LIN {X 0,Y 573.521,Z 573.892,A -85,B 0,C 180,E1 -2263.87,E2 -2263.87} C_VEL
LIN {X 0,Y 573.779,Z 548.951,A -85,B 0,C 180,E1 -2266.545,E2 -2266.545} C_VEL
LIN {X 0,Y 574.092,Z 520.138,A -85,B 0,C 180,E1 -2269.699,E2 -2269.699} C_VEL
LIN {X 0,Y 574.414,Z 495.16,A -85,B 0,C 180,E1 -2272.479,E2 -2272.479} C_VEL
LIN {X 0,Y 574.81,Z 471.063,A -85,B 0,C 180,E1 -2275.207,E2 -2275.207} C_VEL
LIN {X 0,Y 574.89,Z 460.282,A -85,B 0,C 180,E1 -2276.409,E2 -2276.409} C_VEL
LIN {X 0,Y 573.276,Z 453.235,A -85,B 0,C 180,E1 -2277.27,E2 -2277.27} C_VEL
LIN {X 0,Y 573.249,Z 453.075,A -85,B 0,C 180,E1 -2280.175,E2 -2280.175} C_VEL
LIN {X 0,Y 573.254,Z 453.074,A -85,B 0,C 180,E1 -2282.644,E2 -2282.644} C_VEL
LIN {X 0,Y 573.205,Z 453.079,A -85,B 0,C 180,E1 -2285.187,E2 -2285.187} C_VEL
LIN {X 0,Y 573.234,Z 453.078,A -85,B 0,C 180,E1 -2287.807,E2 -2287.807} C_VEL
LIN {X 0,Y 573.266,Z 453.074,A -85,B 0,C 180,E1 -2290.527,E2 -2290.527} C_VEL
LIN {X 0,Y 573.249,Z 453.075,A -85,B 0,C 180,E1 -2293.669,E2 -2293.669} C_VEL
LIN {X 0,Y 573.234,Z 453.076,A -85,B 0,C 180,E1 -2296.64,E2 -2296.64} C_VEL
LIN {X 0,Y 573.268,Z 453.071,A -85,B 0,C 180,E1 -2299.477,E2 -2299.477} C_VEL
LIN {X 0,Y 573.23,Z 453.083,A -85,B 0,C 180,E1 -2302.192,E2 -2302.192} C_VEL
LIN {X 0,Y 573.263,Z 453.073,A -85,B 0,C 180,E1 -2304.816,E2 -2304.816} C_VEL
LIN {X 0,Y 573.249,Z 453.071,A -85,B 0,C 180,E1 -2307.355,E2 -2307.355} C_VEL
LIN {X 0,Y 573.249,Z 453.075,A -85,B 0,C 180,E1 -2309.824,E2 -2309.824} C_VEL
LIN {X 0,Y 573.281,Z 453.076,A -85,B 0,C 180,E1 -2312.235,E2 -2312.235} C_VEL
LIN {X 0,Y 573.261,Z 453.071,A -85,B 0,C 180,E1 -2315.12,E2 -2315.12} C_VEL
LIN {X 0,Y 573.23,Z 453.076,A -85,B 0,C 180,E1 -2317.662,E2 -2317.662} C_VEL
LIN {X 0,Y 573.248,Z 453.073,A -85,B 0,C 180,E1 -2319.923,E2 -2319.923} C_VEL
LIN {X 0,Y 573.253,Z 453.073,A -85,B 0,C 180,E1 -2322.988,E2 -2322.988} C_VEL
LIN {X 0,Y 573.263,Z 453.072,A -85,B 0,C 180,E1 -2325.807,E2 -2325.807} C_VEL
LIN {X 0,Y 573.273,Z 453.074,A -85,B 0,C 180,E1 -2328.734,E2 -2328.734} C_VEL
LIN {X 0,Y 573.298,Z 453.066,A -85,B 0,C 180,E1 -2331.541,E2 -2331.541} C_VEL
LIN {X 0,Y 573.285,Z 453.075,A -85,B 0,C 180,E1 -2334.372,E2 -2334.372} C_VEL
LIN {X 0,Y 573.3,Z 453.067,A -85,B 0,C 180,E1 -2337.892,E2 -2337.892} C_VEL
LIN {X 0,Y 573.33,Z 453.07,A -85,B 0,C 180,E1 -2340.702,E2 -2340.702} C_VEL
LIN {X 0,Y 573.233,Z 453.073,A -85,B 0,C 180,E1 -2343.515,E2 -2343.515} C_VEL
LIN {X 0,Y 573.29,Z 453.067,A -85,B 0,C 180,E1 -2345.628,E2 -2345.628} C_VEL
LIN {X 0,Y 573.299,Z 453.073,A -85,B 0,C 180,E1 -2348.459,E2 -2348.459} C_VEL
LIN {X 0,Y 573.289,Z 453.069,A -85,B 0,C 180,E1 -2351.312,E2 -2351.312} C_VEL
LIN {X 0,Y 573.271,Z 453.075,A -85,B 0,C 180,E1 -2354.425,E2 -2354.425} C_VEL
LIN {X 0,Y 573.251,Z 453.076,A -85,B 0,C 180,E1 -2357.112,E2 -2357.112} C_VEL
LIN {X 0,Y 573.249,Z 453.074,A -85,B 0,C 180,E1 -2360.077,E2 -2360.077} C_VEL
LIN {X 0,Y 573.231,Z 453.077,A -85,B 0,C 180,E1 -2362.338,E2 -2362.338} C_VEL
LIN {X 0,Y 573.244,Z 453.077,A -85,B 0,C 180,E1 -2364.403,E2 -2364.403} C_VEL
LIN {X 0,Y 572.618,Z 453.162,A -85,B 0,C 180,E1 -2364.99,E2 -2364.99} C_VEL
LIN {X 0,Y 569.779,Z 453.515,A -85,B 0,C 180,E1 -2365.942,E2 -2365.942} C_VEL
LIN {X 0,Y 567.35,Z 453.816,A -85,B 0,C 180,E1 -2366.708,E2 -2366.708} C_VEL
LIN {X 0,Y 566.298,Z 453.94,A -85,B 0,C 180,E1 -2367.299,E2 -2367.299} C_VEL
LIN {X 0,Y 566.209,Z 453.949,A -85,B 0,C 180,E1 -2367.499,E2 -2367.499} C_VEL
LIN {X 0,Y 566.187,Z 453.953,A -85,B 0,C 180,E1 -2370.593,E2 -2370.593} C_VEL
LIN {X 0,Y 566.222,Z 453.953,A -85,B 0,C 180,E1 -2373.102,E2 -2373.102} C_VEL
LIN {X 0,Y 566.208,Z 453.95,A -85,B 0,C 180,E1 -2375.689,E2 -2375.689} C_VEL
LIN {X 0,Y 566.212,Z 453.952,A -85,B 0,C 180,E1 -2378.56,E2 -2378.56} C_VEL
LIN {X 0,Y 566.207,Z 453.955,A -85,B 0,C 180,E1 -2381.137,E2 -2381.137} C_VEL
LIN {X 0,Y 566.196,Z 453.951,A -85,B 0,C 180,E1 -2384.036,E2 -2384.036} C_VEL
LIN {X 0,Y 566.207,Z 453.955,A -85,B 0,C 180,E1 -2387.083,E2 -2387.083} C_VEL
LIN {X 0,Y 566.225,Z 453.948,A -85,B 0,C 180,E1 -2389.804,E2 -2389.804} C_VEL
LIN {X 0,Y 566.198,Z 453.954,A -85,B 0,C 180,E1 -2392.6,E2 -2392.6} C_VEL
LIN {X 0,Y 566.212,Z 453.947,A -85,B 0,C 180,E1 -2395.183,E2 -2395.183} C_VEL
LIN {X 0,Y 566.234,Z 453.947,A -85,B 0,C 180,E1 -2397.745,E2 -2397.745} C_VEL
LIN {X 0,Y 566.204,Z 453.952,A -85,B 0,C 180,E1 -2400.329,E2 -2400.329} C_VEL
LIN {X 0,Y 566.212,Z 453.949,A -85,B 0,C 180,E1 -2402.662,E2 -2402.662} C_VEL
LIN {X 0,Y 566.238,Z 453.954,A -85,B 0,C 180,E1 -2405.04,E2 -2405.04} C_VEL
LIN {X 0,Y 566.196,Z 453.949,A -85,B 0,C 180,E1 -2408.138,E2 -2408.138} C_VEL
LIN {X 0,Y 566.239,Z 453.949,A -85,B 0,C 180,E1 -2410.612,E2 -2410.612} C_VEL
LIN {X 0,Y 566.218,Z 453.944,A -85,B 0,C 180,E1 -2413.413,E2 -2413.413} C_VEL
LIN {X 0,Y 566.282,Z 454.118,A -85,B 0,C 180,E1 -2416.293,E2 -2416.293} C_VEL
LIN {X 0,Y 566.5,Z 455.143,A -85,B 0,C 180,E1 -2416.407,E2 -2416.407} C_VEL
LIN {X 0,Y 567.065,Z 456.976,A -85,B 0,C 180,E1 -2416.453,E2 -2416.453} C_VEL
LIN {X 0,Y 566.992,Z 533.99,A -85,B 0,C 180,E1 -2417.45,E2 -2417.45} C_VEL
LIN {X 0,Y 566.878,Z 547.245,A -85,B 0,C 180,E1 -2417.765,E2 -2417.765} C_VEL
LIN {X 0,Y 566.749,Z 559.399,A -85,B 0,C 180,E1 -2418.194,E2 -2418.194} C_VEL
LIN {X 0,Y 566.633,Z 571.542,A -85,B 0,C 180,E1 -2418.776,E2 -2418.776} C_VEL
LIN {X 0,Y 566.459,Z 582.558,A -85,B 0,C 180,E1 -2419.456,E2 -2419.456} C_VEL
LIN {X 0,Y 566.323,Z 593.075,A -85,B 0,C 180,E1 -2420.266,E2 -2420.266} C_VEL
LIN {X 0,Y 566.221,Z 601.673,A -85,B 0,C 180,E1 -2421.075,E2 -2421.075} C_VEL
LIN {X 0,Y 566.113,Z 609.593,A -85,B 0,C 180,E1 -2421.972,E2 -2421.972} C_VEL
LIN {X 0,Y 566.05,Z 616.16,A -85,B 0,C 180,E1 -2422.868,E2 -2422.868} C_VEL
LIN {X 0,Y 566.003,Z 622.629,A -85,B 0,C 180,E1 -2423.942,E2 -2423.942} C_VEL
LIN {X 0,Y 565.878,Z 627.766,A -85,B 0,C 180,E1 -2425.013,E2 -2425.013} C_VEL
LIN {X 0,Y 565.926,Z 631.754,A -85,B 0,C 180,E1 -2426.084,E2 -2426.084} C_VEL
LIN {X 0,Y 565.877,Z 634.704,A -85,B 0,C 180,E1 -2427.153,E2 -2427.153} C_VEL
LIN {X 0,Y 565.84,Z 636.128,A -85,B 0,C 180,E1 -2427.865,E2 -2427.865} C_VEL
LIN {X 0,Y 565.841,Z 637.756,A -85,B 0,C 180,E1 -2429.288,E2 -2429.288} C_VEL
LIN {X 0,Y 565.839,Z 637.996,A -85,B 0,C 180,E1 -2430,E2 -2430} C_VEL
LIN {X 0,Y 565.841,Z 637.815,A -85,B 0,C 180,E1 -2430.712,E2 -2430.712} C_VEL
LIN {X 0,Y 565.84,Z 636.269,A -85,B 0,C 180,E1 -2432.135,E2 -2432.135} C_VEL
LIN {X 0,Y 565.878,Z 634.909,A -85,B 0,C 180,E1 -2432.847,E2 -2432.847} C_VEL
LIN {X 0,Y 565.927,Z 632.029,A -85,B 0,C 180,E1 -2433.916,E2 -2433.916} C_VEL
LIN {X 0,Y 565.878,Z 628.129,A -85,B 0,C 180,E1 -2434.987,E2 -2434.987} C_VEL
LIN {X 0,Y 565.99,Z 623.098,A -85,B 0,C 180,E1 -2436.058,E2 -2436.058} C_VEL
LIN {X 0,Y 566.031,Z 616.774,A -85,B 0,C 180,E1 -2437.132,E2 -2437.132} C_VEL
LIN {X 0,Y 566.133,Z 608.85,A -85,B 0,C 180,E1 -2438.207,E2 -2438.207} C_VEL
LIN {X 0,Y 566.249,Z 598.998,A -85,B 0,C 180,E1 -2439.285,E2 -2439.285} C_VEL
LIN {X 0,Y 566.423,Z 588.683,A -85,B 0,C 180,E1 -2440.184,E2 -2440.184} C_VEL
LIN {X 0,Y 566.581,Z 577.399,A -85,B 0,C 180,E1 -2440.971,E2 -2440.971} C_VEL
LIN {X 0,Y 566.679,Z 565.488,A -85,B 0,C 180,E1 -2441.626,E2 -2441.626} C_VEL
LIN {X 0,Y 566.819,Z 553.476,A -85,B 0,C 180,E1 -2442.122,E2 -2442.122} C_VEL
LIN {X 0,Y 566.936,Z 540.434,A -85,B 0,C 180,E1 -2442.506,E2 -2442.506} C_VEL
LIN {X 0,Y 567.025,Z 528.072,A -85,B 0,C 180,E1 -2442.732,E2 -2442.732} C_VEL
LIN {X 0,Y 566.994,Z 456.838,A -85,B 0,C 180,E1 -2443.64,E2 -2443.64} C_VEL
LIN {X 0,Y 566.421,Z 454.812,A -85,B 0,C 180,E1 -2443.704,E2 -2443.704} C_VEL
LIN {X 0,Y 566.255,Z 453.999,A -85,B 0,C 180,E1 -2443.845,E2 -2443.845} C_VEL
LIN {X 0,Y 566.227,Z 453.941,A -85,B 0,C 180,E1 -2447.113,E2 -2447.113} C_VEL
LIN {X 0,Y 566.214,Z 453.951,A -85,B 0,C 180,E1 -2449.58,E2 -2449.58} C_VEL
LIN {X 0,Y 566.195,Z 453.949,A -85,B 0,C 180,E1 -2451.862,E2 -2451.862} C_VEL
LIN {X 0,Y 566.219,Z 453.956,A -85,B 0,C 180,E1 -2455.029,E2 -2455.029} C_VEL
LIN {X 0,Y 566.212,Z 453.95,A -85,B 0,C 180,E1 -2457.338,E2 -2457.338} C_VEL
LIN {X 0,Y 566.202,Z 453.951,A -85,B 0,C 180,E1 -2459.768,E2 -2459.768} C_VEL
LIN {X 0,Y 566.206,Z 453.951,A -85,B 0,C 180,E1 -2462.43,E2 -2462.43} C_VEL
LIN {X 0,Y 566.199,Z 453.961,A -85,B 0,C 180,E1 -2464.992,E2 -2464.992} C_VEL
LIN {X 0,Y 566.195,Z 453.954,A -85,B 0,C 180,E1 -2467.46,E2 -2467.46} C_VEL
LIN {X 0,Y 566.225,Z 453.948,A -85,B 0,C 180,E1 -2470.196,E2 -2470.196} C_VEL
LIN {X 0,Y 566.202,Z 453.956,A -85,B 0,C 180,E1 -2473.053,E2 -2473.053} C_VEL
LIN {X 0,Y 566.194,Z 453.952,A -85,B 0,C 180,E1 -2476.048,E2 -2476.048} C_VEL
LIN {X 0,Y 566.207,Z 453.954,A -85,B 0,C 180,E1 -2478.863,E2 -2478.863} C_VEL
LIN {X 0,Y 566.185,Z 453.954,A -85,B 0,C 180,E1 -2481.637,E2 -2481.637} C_VEL
LIN {X 0,Y 566.208,Z 453.95,A -85,B 0,C 180,E1 -2484.311,E2 -2484.311} C_VEL
LIN {X 0,Y 566.222,Z 453.952,A -85,B 0,C 180,E1 -2486.898,E2 -2486.898} C_VEL
LIN {X 0,Y 566.187,Z 453.954,A -85,B 0,C 180,E1 -2489.407,E2 -2489.407} C_VEL
LIN {X 0,Y 566.22,Z 453.948,A -85,B 0,C 180,E1 -2491.858,E2 -2491.858} C_VEL
LIN {X 0,Y 566.219,Z 453.948,A -85,B 0,C 180,E1 -2494.251,E2 -2494.251} C_VEL
LIN {X 0,Y 566.184,Z 453.954,A -85,B 0,C 180,E1 -2496.713,E2 -2496.713} C_VEL
LIN {X 0,Y 566.212,Z 453.954,A -85,B 0,C 180,E1 -2499.663,E2 -2499.663} C_VEL
LIN {X 0,Y 566.195,Z 453.952,A -85,B 0,C 180,E1 -2502.668,E2 -2502.668} C_VEL
LIN {X 0,Y 566.223,Z 453.953,A -85,B 0,C 180,E1 -2505.626,E2 -2505.626} C_VEL
LIN {X 0,Y 566.265,Z 453.943,A -85,B 0,C 180,E1 -2508.654,E2 -2508.654} C_VEL
LIN {X 0,Y 566.241,Z 453.954,A -85,B 0,C 180,E1 -2511.434,E2 -2511.434} C_VEL
LIN {X 0,Y 566.252,Z 453.944,A -85,B 0,C 180,E1 -2514.302,E2 -2514.302} C_VEL
LIN {X 0,Y 566.271,Z 453.943,A -85,B 0,C 180,E1 -2517.866,E2 -2517.866} C_VEL
LIN {X 0,Y 566.298,Z 453.939,A -85,B 0,C 180,E1 -2520.711,E2 -2520.711} C_VEL
LIN {X 0,Y 566.271,Z 453.942,A -85,B 0,C 180,E1 -2522.846,E2 -2522.846} C_VEL
LIN {X 0,Y 566.252,Z 453.95,A -85,B 0,C 180,E1 -2525.698,E2 -2525.698} C_VEL
LIN {X 0,Y 566.239,Z 453.945,A -85,B 0,C 180,E1 -2528.566,E2 -2528.566} C_VEL
LIN {X 0,Y 566.241,Z 453.952,A -85,B 0,C 180,E1 -2531.454,E2 -2531.454} C_VEL
LIN {X 0,Y 566.223,Z 453.948,A -85,B 0,C 180,E1 -2534.507,E2 -2534.507} C_VEL
LIN {X 0,Y 566.195,Z 453.956,A -85,B 0,C 180,E1 -2537.332,E2 -2537.332} C_VEL
LIN {X 0,Y 566.211,Z 453.948,A -85,B 0,C 180,E1 -2540.337,E2 -2540.337} C_VEL
LIN {X 0,Y 566.181,Z 453.96,A -85,B 0,C 180,E1 -2543.404,E2 -2543.404} C_VEL
LIN {X 0,Y 566.218,Z 453.953,A -85,B 0,C 180,E1 -2545.749,E2 -2545.749} C_VEL
LIN {X 0,Y 566.199,Z 453.952,A -85,B 0,C 180,E1 -2548.204,E2 -2548.204} C_VEL
LIN {X 0,Y 566.186,Z 453.953,A -85,B 0,C 180,E1 -2550.593,E2 -2550.593} C_VEL
LIN {X 0,Y 566.222,Z 453.948,A -85,B 0,C 180,E1 -2553.102,E2 -2553.102} C_VEL
LIN {X 0,Y 566.207,Z 453.96,A -85,B 0,C 180,E1 -2555.689,E2 -2555.689} C_VEL
LIN {X 0,Y 566.21,Z 453.949,A -85,B 0,C 180,E1 -2558.56,E2 -2558.56} C_VEL
LIN {X 0,Y 566.206,Z 453.952,A -85,B 0,C 180,E1 -2561.137,E2 -2561.137} C_VEL
LIN {X 0,Y 566.192,Z 453.955,A -85,B 0,C 180,E1 -2564.036,E2 -2564.036} C_VEL
LIN {X 0,Y 566.201,Z 453.952,A -85,B 0,C 180,E1 -2567.083,E2 -2567.083} C_VEL
LIN {X 0,Y 566.224,Z 453.954,A -85,B 0,C 180,E1 -2569.804,E2 -2569.804} C_VEL
LIN {X 0,Y 566.197,Z 453.951,A -85,B 0,C 180,E1 -2572.6,E2 -2572.6} C_VEL
LIN {X 0,Y 566.205,Z 453.952,A -85,B 0,C 180,E1 -2575.183,E2 -2575.183} C_VEL
LIN {X 0,Y 566.233,Z 453.955,A -85,B 0,C 180,E1 -2577.744,E2 -2577.744} C_VEL
LIN {X 0,Y 566.203,Z 453.95,A -85,B 0,C 180,E1 -2580.329,E2 -2580.329} C_VEL
LIN {X 0,Y 566.238,Z 454.137,A -85,B 0,C 180,E1 -2582.563,E2 -2582.563} C_VEL
LIN {X 0,Y 568.003,Z 462.182,A -85,B 0,C 180,E1 -2583.55,E2 -2583.55} C_VEL
LIN {X 0,Y 567.78,Z 486.01,A -85,B 0,C 180,E1 -2586.194,E2 -2586.194} C_VEL
LIN {X 0,Y 567.361,Z 510.289,A -85,B 0,C 180,E1 -2588.948,E2 -2588.948} C_VEL
LIN {X 0,Y 566.973,Z 537.184,A -85,B 0,C 180,E1 -2591.948,E2 -2591.948} C_VEL
LIN {X 0,Y 566.679,Z 562.399,A -85,B 0,C 180,E1 -2594.72,E2 -2594.72} C_VEL
LIN {X 0,Y 566.56,Z 573.901,A -85,B 0,C 180,E1 -2595.956,E2 -2595.956} C_VEL
LIN {X 0,Y 567.212,Z 579.746,A -85,B 0,C 180,E1 -2596.064,E2 -2596.064} C_VEL
LIN {X 0,Y 566.975,Z 683.962,A -85,B 0,C 180,E1 -2597.404,E2 -2597.404} C_VEL
LIN {X 0,Y 566.891,Z 696.467,A -85,B 0,C 180,E1 -2597.697,E2 -2597.697} C_VEL
LIN {X 0,Y 566.745,Z 708.925,A -85,B 0,C 180,E1 -2598.13,E2 -2598.13} C_VEL
LIN {X 0,Y 566.627,Z 721.167,A -85,B 0,C 180,E1 -2598.709,E2 -2598.709} C_VEL
LIN {X 0,Y 566.459,Z 733.205,A -85,B 0,C 180,E1 -2599.456,E2 -2599.456} C_VEL
LIN {X 0,Y 566.319,Z 743.604,A -85,B 0,C 180,E1 -2600.266,E2 -2600.266} C_VEL
LIN {X 0,Y 566.207,Z 752.115,A -85,B 0,C 180,E1 -2601.074,E2 -2601.074} C_VEL
LIN {X 0,Y 566.112,Z 759.962,A -85,B 0,C 180,E1 -2601.972,E2 -2601.972} C_VEL
LIN {X 0,Y 566.003,Z 767.623,A -85,B 0,C 180,E1 -2603.047,E2 -2603.047} C_VEL
LIN {X 0,Y 566.004,Z 774.681,A -85,B 0,C 180,E1 -2604.299,E2 -2604.299} C_VEL
LIN {X 0,Y 565.933,Z 779.372,A -85,B 0,C 180,E1 -2605.37,E2 -2605.37} C_VEL
LIN {X 0,Y 565.927,Z 782.958,A -85,B 0,C 180,E1 -2606.44,E2 -2606.44} C_VEL
LIN {X 0,Y 565.878,Z 784.808,A -85,B 0,C 180,E1 -2607.153,E2 -2607.153} C_VEL
LIN {X 0,Y 565.846,Z 787.186,A -85,B 0,C 180,E1 -2608.577,E2 -2608.577} C_VEL
LIN {X 0,Y 565.839,Z 788,A -85,B 0,C 180,E1 -2610,E2 -2610} C_VEL
LIN {X 0,Y 565.846,Z 787.186,A -85,B 0,C 180,E1 -2611.423,E2 -2611.423} C_VEL
LIN {X 0,Y 565.878,Z 784.81,A -85,B 0,C 180,E1 -2612.847,E2 -2612.847} C_VEL
LIN {X 0,Y 565.926,Z 781.896,A -85,B 0,C 180,E1 -2613.916,E2 -2613.916} C_VEL
LIN {X 0,Y 565.878,Z 777.949,A -85,B 0,C 180,E1 -2614.987,E2 -2614.987} C_VEL
LIN {X 0,Y 566.002,Z 772.867,A -85,B 0,C 180,E1 -2616.058,E2 -2616.058} C_VEL
LIN {X 0,Y 566.04,Z 766.47,A -85,B 0,C 180,E1 -2617.132,E2 -2617.132} C_VEL
LIN {X 0,Y 566.133,Z 758.48,A -85,B 0,C 180,E1 -2618.207,E2 -2618.207} C_VEL
LIN {X 0,Y 566.228,Z 750.338,A -85,B 0,C 180,E1 -2619.105,E2 -2619.105} C_VEL
LIN {X 0,Y 566.339,Z 740.404,A -85,B 0,C 180,E1 -2620.005,E2 -2620.005} C_VEL
LIN {X 0,Y 566.526,Z 729.287,A -85,B 0,C 180,E1 -2620.807,E2 -2620.807} C_VEL
LIN {X 0,Y 566.66,Z 718.182,A -85,B 0,C 180,E1 -2621.445,E2 -2621.445} C_VEL
LIN {X 0,Y 566.743,Z 705.991,A -85,B 0,C 180,E1 -2621.988,E2 -2621.988} C_VEL
LIN {X 0,Y 566.903,Z 693.188,A -85,B 0,C 180,E1 -2622.393,E2 -2622.393} C_VEL
LIN {X 0,Y 566.991,Z 679.622,A -85,B 0,C 180,E1 -2622.664,E2 -2622.664} C_VEL
LIN {X 0,Y 567.072,Z 577.956,A -85,B 0,C 180,E1 -2623.962,E2 -2623.962} C_VEL
LIN {X 0,Y 566.566,Z 573.899,A -85,B 0,C 180,E1 -2624.043,E2 -2624.043} C_VEL
LIN {X 0,Y 566.841,Z 547.449,A -85,B 0,C 180,E1 -2626.919,E2 -2626.919} C_VEL
LIN {X 0,Y 567.214,Z 520.711,A -85,B 0,C 180,E1 -2629.883,E2 -2629.883} C_VEL
LIN {X 0,Y 567.67,Z 493.479,A -85,B 0,C 180,E1 -2632.953,E2 -2632.953} C_VEL
LIN {X 0,Y 567.919,Z 474.04,A -85,B 0,C 180,E1 -2635.135,E2 -2635.135} C_VEL
LIN {X 0,Y 567.848,Z 461.024,A -85,B 0,C 180,E1 -2636.584,E2 -2636.584} C_VEL
LIN {X 0,Y 566.228,Z 454.041,A -85,B 0,C 180,E1 -2637.463,E2 -2637.463} C_VEL
LIN {X 0,Y 566.187,Z 453.955,A -85,B 0,C 180,E1 -2640.592,E2 -2640.592} C_VEL
LIN {X 0,Y 566.219,Z 453.948,A -85,B 0,C 180,E1 -2643.101,E2 -2643.101} C_VEL
LIN {X 0,Y 566.16,Z 453.96,A -85,B 0,C 180,E1 -2645.691,E2 -2645.691} C_VEL
LIN {X 0,Y 566.214,Z 453.953,A -85,B 0,C 180,E1 -2648.558,E2 -2648.558} C_VEL
LIN {X 0,Y 566.208,Z 453.948,A -85,B 0,C 180,E1 -2651.135,E2 -2651.135} C_VEL
LIN {X 0,Y 566.196,Z 453.959,A -85,B 0,C 180,E1 -2654.035,E2 -2654.035} C_VEL
LIN {X 0,Y 566.196,Z 453.949,A -85,B 0,C 180,E1 -2657.082,E2 -2657.082} C_VEL
LIN {X 0,Y 566.221,Z 453.951,A -85,B 0,C 180,E1 -2659.802,E2 -2659.802} C_VEL
LIN {X 0,Y 566.192,Z 453.957,A -85,B 0,C 180,E1 -2662.598,E2 -2662.598} C_VEL
LIN {X 0,Y 566.215,Z 453.948,A -85,B 0,C 180,E1 -2665.182,E2 -2665.182} C_VEL
LIN {X 0,Y 566.228,Z 453.947,A -85,B 0,C 180,E1 -2667.743,E2 -2667.743} C_VEL
LIN {X 0,Y 566.221,Z 453.958,A -85,B 0,C 180,E1 -2670.323,E2 -2670.323} C_VEL
LIN {X 0,Y 566.226,Z 453.944,A -85,B 0,C 180,E1 -2673.334,E2 -2673.334} C_VEL
LIN {X 0,Y 566.19,Z 453.953,A -85,B 0,C 180,E1 -2675.819,E2 -2675.819} C_VEL
LIN {X 0,Y 566.208,Z 453.951,A -85,B 0,C 180,E1 -2678.902,E2 -2678.902} C_VEL
LIN {X 0,Y 566.204,Z 453.946,A -85,B 0,C 180,E1 -2681.172,E2 -2681.172} C_VEL
LIN {X 0,Y 566.212,Z 453.948,A -85,B 0,C 180,E1 -2683.412,E2 -2683.412} C_VEL
LIN {X 0,Y 566.191,Z 453.96,A -85,B 0,C 180,E1 -2686.359,E2 -2686.359} C_VEL
LIN {X 0,Y 566.265,Z 453.949,A -85,B 0,C 180,E1 -2688.654,E2 -2688.654} C_VEL
LIN {X 0,Y 566.239,Z 453.946,A -85,B 0,C 180,E1 -2691.434,E2 -2691.434} C_VEL
LIN {X 0,Y 566.253,Z 453.95,A -85,B 0,C 180,E1 -2694.302,E2 -2694.302} C_VEL
LIN {X 0,Y 566.272,Z 453.942,A -85,B 0,C 180,E1 -2697.866,E2 -2697.866} C_VEL
LIN {X 0,Y 566.3,Z 453.945,A -85,B 0,C 180,E1 -2700.711,E2 -2700.711} C_VEL
LIN {X 0,Y 566.272,Z 453.947,A -85,B 0,C 180,E1 -2702.846,E2 -2702.846} C_VEL
LIN {X 0,Y 566.258,Z 453.943,A -85,B 0,C 180,E1 -2705.698,E2 -2705.698} C_VEL
LIN {X 0,Y 566.24,Z 453.954,A -85,B 0,C 180,E1 -2708.566,E2 -2708.566} C_VEL
LIN {X 0,Y 566.241,Z 453.946,A -85,B 0,C 180,E1 -2711.454,E2 -2711.454} C_VEL
LIN {X 0,Y 566.224,Z 453.954,A -85,B 0,C 180,E1 -2714.507,E2 -2714.507} C_VEL
LIN {X 0,Y 566.195,Z 453.952,A -85,B 0,C 180,E1 -2717.332,E2 -2717.332} C_VEL
LIN {X 0,Y 566.212,Z 453.953,A -85,B 0,C 180,E1 -2720.337,E2 -2720.337} C_VEL
LIN {X 0,Y 566.182,Z 453.954,A -85,B 0,C 180,E1 -2723.404,E2 -2723.404} C_VEL
LIN {X 0,Y 566.219,Z 453.948,A -85,B 0,C 180,E1 -2725.749,E2 -2725.749} C_VEL
LIN {X 0,Y 566.209,Z 453.949,A -85,B 0,C 180,E1 -2727.499,E2 -2727.499} C_VEL
LIN {X 0,Y 565.531,Z 454.034,A -85,B 0,C 180,E1 -2728.093,E2 -2728.093} C_VEL
LIN {X 0,Y 562.667,Z 454.391,A -85,B 0,C 180,E1 -2729.057,E2 -2729.057} C_VEL
LIN {X 0,Y 560.255,Z 454.687,A -85,B 0,C 180,E1 -2729.832,E2 -2729.832} C_VEL
LIN {X 0,Y 559.227,Z 454.817,A -85,B 0,C 180,E1 -2730.431,E2 -2730.431} C_VEL
LIN {X 0,Y 559.146,Z 454.826,A -85,B 0,C 180,E1 -2730.634,E2 -2730.634} C_VEL
LIN {X 0,Y 559.171,Z 454.826,A -85,B 0,C 180,E1 -2733.575,E2 -2733.575} C_VEL
LIN {X 0,Y 559.164,Z 454.831,A -85,B 0,C 180,E1 -2736.449,E2 -2736.449} C_VEL
LIN {X 0,Y 559.174,Z 454.83,A -85,B 0,C 180,E1 -2738.934,E2 -2738.934} C_VEL
LIN {X 0,Y 559.187,Z 454.823,A -85,B 0,C 180,E1 -2741.768,E2 -2741.768} C_VEL
LIN {X 0,Y 559.136,Z 454.837,A -85,B 0,C 180,E1 -2744.74,E2 -2744.74} C_VEL
LIN {X 0,Y 559.165,Z 454.83,A -85,B 0,C 180,E1 -2747.258,E2 -2747.258} C_VEL
LIN {X 0,Y 559.184,Z 454.825,A -85,B 0,C 180,E1 -2750.136,E2 -2750.136} C_VEL
LIN {X 0,Y 559.144,Z 454.837,A -85,B 0,C 180,E1 -2752.893,E2 -2752.893} C_VEL
LIN {X 0,Y 559.166,Z 454.818,A -85,B 0,C 180,E1 -2756.051,E2 -2756.051} C_VEL
LIN {X 0,Y 559.164,Z 454.835,A -85,B 0,C 180,E1 -2758.982,E2 -2758.982} C_VEL
LIN {X 0,Y 559.169,Z 454.825,A -85,B 0,C 180,E1 -2761.619,E2 -2761.619} C_VEL
LIN {X 0,Y 559.182,Z 454.824,A -85,B 0,C 180,E1 -2763.904,E2 -2763.904} C_VEL
LIN {X 0,Y 559.144,Z 454.832,A -85,B 0,C 180,E1 -2766.571,E2 -2766.571} C_VEL
LIN {X 0,Y 559.183,Z 454.832,A -85,B 0,C 180,E1 -2769.396,E2 -2769.396} C_VEL
LIN {X 0,Y 559.149,Z 454.822,A -85,B 0,C 180,E1 -2771.686,E2 -2771.686} C_VEL
LIN {X 0,Y 559.17,Z 454.828,A -85,B 0,C 180,E1 -2773.948,E2 -2773.948} C_VEL
LIN {X 0,Y 559.26,Z 454.984,A -85,B 0,C 180,E1 -2776.117,E2 -2776.117} C_VEL
LIN {X 0,Y 559.47,Z 456.08,A -85,B 0,C 180,E1 -2776.237,E2 -2776.237} C_VEL
LIN {X 0,Y 560.271,Z 458.975,A -85,B 0,C 180,E1 -2776.305,E2 -2776.305} C_VEL
LIN {X 0,Y 560.089,Z 534.259,A -85,B 0,C 180,E1 -2777.292,E2 -2777.292} C_VEL
LIN {X 0,Y 559.937,Z 547.456,A -85,B 0,C 180,E1 -2777.611,E2 -2777.611} C_VEL
LIN {X 0,Y 559.798,Z 559.52,A -85,B 0,C 180,E1 -2778.045,E2 -2778.045} C_VEL
LIN {X 0,Y 559.648,Z 571.091,A -85,B 0,C 180,E1 -2778.607,E2 -2778.607} C_VEL
LIN {X 0,Y 559.482,Z 582.563,A -85,B 0,C 180,E1 -2779.323,E2 -2779.323} C_VEL
LIN {X 0,Y 559.304,Z 593.08,A -85,B 0,C 180,E1 -2780.142,E2 -2780.142} C_VEL
LIN {X 0,Y 559.197,Z 601.678,A -85,B 0,C 180,E1 -2780.962,E2 -2780.962} C_VEL
LIN {X 0,Y 559.05,Z 609.597,A -85,B 0,C 180,E1 -2781.87,E2 -2781.87} C_VEL
LIN {X 0,Y 558.971,Z 617.457,A -85,B 0,C 180,E1 -2782.977,E2 -2782.977} C_VEL
LIN {X 0,Y 558.936,Z 624.456,A -85,B 0,C 180,E1 -2784.227,E2 -2784.227} C_VEL
LIN {X 0,Y 558.826,Z 629.197,A -85,B 0,C 180,E1 -2785.311,E2 -2785.311} C_VEL
LIN {X 0,Y 558.836,Z 632.828,A -85,B 0,C 180,E1 -2786.395,E2 -2786.395} C_VEL
LIN {X 0,Y 558.799,Z 634.706,A -85,B 0,C 180,E1 -2787.116,E2 -2787.116} C_VEL
LIN {X 0,Y 558.746,Z 636.128,A -85,B 0,C 180,E1 -2787.838,E2 -2787.838} C_VEL
LIN {X 0,Y 558.741,Z 637.756,A -85,B 0,C 180,E1 -2789.279,E2 -2789.279} C_VEL
LIN {X 0,Y 558.74,Z 637.996,A -85,B 0,C 180,E1 -2790,E2 -2790} C_VEL
LIN {X 0,Y 558.741,Z 637.815,A -85,B 0,C 180,E1 -2790.721,E2 -2790.721} C_VEL
LIN {X 0,Y 558.746,Z 636.268,A -85,B 0,C 180,E1 -2792.162,E2 -2792.162} C_VEL
LIN {X 0,Y 558.8,Z 634.907,A -85,B 0,C 180,E1 -2792.884,E2 -2792.884} C_VEL
LIN {X 0,Y 558.844,Z 632.027,A -85,B 0,C 180,E1 -2793.966,E2 -2793.966} C_VEL
LIN {X 0,Y 558.798,Z 628.127,A -85,B 0,C 180,E1 -2795.051,E2 -2795.051} C_VEL
LIN {X 0,Y 558.91,Z 623.095,A -85,B 0,C 180,E1 -2796.136,E2 -2796.136} C_VEL
LIN {X 0,Y 558.972,Z 616.77,A -85,B 0,C 180,E1 -2797.223,E2 -2797.223} C_VEL
LIN {X 0,Y 559.096,Z 608.846,A -85,B 0,C 180,E1 -2798.311,E2 -2798.311} C_VEL
LIN {X 0,Y 559.182,Z 600.775,A -85,B 0,C 180,E1 -2799.221,E2 -2799.221} C_VEL
LIN {X 0,Y 559.355,Z 590.925,A -85,B 0,C 180,E1 -2800.131,E2 -2800.131} C_VEL
LIN {X 0,Y 559.581,Z 580.09,A -85,B 0,C 180,E1 -2800.937,E2 -2800.937} C_VEL
LIN {X 0,Y 559.665,Z 568.425,A -85,B 0,C 180,E1 -2801.624,E2 -2801.624} C_VEL
LIN {X 0,Y 559.82,Z 556.436,A -85,B 0,C 180,E1 -2802.171,E2 -2802.171} C_VEL
LIN {X 0,Y 559.991,Z 544.28,A -85,B 0,C 180,E1 -2802.572,E2 -2802.572} C_VEL
LIN {X 0,Y 560.108,Z 532.804,A -85,B 0,C 180,E1 -2802.822,E2 -2802.822} C_VEL
LIN {X 0,Y 560.11,Z 458.096,A -85,B 0,C 180,E1 -2803.801,E2 -2803.801} C_VEL
LIN {X 0,Y 559.365,Z 455.639,A -85,B 0,C 180,E1 -2803.88,E2 -2803.88} C_VEL
LIN {X 0,Y 559.217,Z 454.869,A -85,B 0,C 180,E1 -2804.023,E2 -2804.023} C_VEL
LIN {X 0,Y 559.174,Z 454.817,A -85,B 0,C 180,E1 -2807.213,E2 -2807.213} C_VEL
LIN {X 0,Y 559.175,Z 454.827,A -85,B 0,C 180,E1 -2809.837,E2 -2809.837} C_VEL
LIN {X 0,Y 559.143,Z 454.828,A -85,B 0,C 180,E1 -2812.152,E2 -2812.152} C_VEL
LIN {X 0,Y 559.177,Z 454.829,A -85,B 0,C 180,E1 -2815.297,E2 -2815.297} C_VEL
LIN {X 0,Y 559.158,Z 454.825,A -85,B 0,C 180,E1 -2817.713,E2 -2817.713} C_VEL
LIN {X 0,Y 559.157,Z 454.829,A -85,B 0,C 180,E1 -2820.182,E2 -2820.182} C_VEL
LIN {X 0,Y 559.173,Z 454.83,A -85,B 0,C 180,E1 -2822.713,E2 -2822.713} C_VEL
LIN {X 0,Y 559.142,Z 454.834,A -85,B 0,C 180,E1 -2825.322,E2 -2825.322} C_VEL
LIN {X 0,Y 559.134,Z 454.83,A -85,B 0,C 180,E1 -2828.016,E2 -2828.016} C_VEL
LIN {X 0,Y 559.174,Z 454.832,A -85,B 0,C 180,E1 -2830.81,E2 -2830.81} C_VEL
LIN {X 0,Y 559.159,Z 454.828,A -85,B 0,C 180,E1 -2833.731,E2 -2833.731} C_VEL
LIN {X 0,Y 559.142,Z 454.835,A -85,B 0,C 180,E1 -2836.803,E2 -2836.803} C_VEL
LIN {X 0,Y 559.171,Z 454.829,A -85,B 0,C 180,E1 -2839.189,E2 -2839.189} C_VEL
LIN {X 0,Y 559.13,Z 454.83,A -85,B 0,C 180,E1 -2841.982,E2 -2841.982} C_VEL
LIN {X 0,Y 559.155,Z 454.832,A -85,B 0,C 180,E1 -2844.782,E2 -2844.782} C_VEL
LIN {X 0,Y 559.168,Z 454.829,A -85,B 0,C 180,E1 -2847.361,E2 -2847.361} C_VEL
LIN {X 0,Y 559.182,Z 454.818,A -85,B 0,C 180,E1 -2850.134,E2 -2850.134} C_VEL
LIN {X 0,Y 559.175,Z 454.833,A -85,B 0,C 180,E1 -2853.169,E2 -2853.169} C_VEL
LIN {X 0,Y 559.149,Z 454.835,A -85,B 0,C 180,E1 -2855.494,E2 -2855.494} C_VEL
LIN {X 0,Y 559.168,Z 454.826,A -85,B 0,C 180,E1 -2858.624,E2 -2858.624} C_VEL
LIN {X 0,Y 559.163,Z 454.831,A -85,B 0,C 180,E1 -2860.926,E2 -2860.926} C_VEL
LIN {X 0,Y 559.162,Z 454.827,A -85,B 0,C 180,E1 -2863.948,E2 -2863.948} C_VEL
LIN {X 0,Y 559.164,Z 454.827,A -85,B 0,C 180,E1 -2866.184,E2 -2866.184} C_VEL
LIN {X 0,Y 559.201,Z 454.828,A -85,B 0,C 180,E1 -2869.134,E2 -2869.134} C_VEL
LIN {X 0,Y 559.201,Z 454.823,A -85,B 0,C 180,E1 -2872.054,E2 -2872.054} C_VEL
LIN {X 0,Y 559.252,Z 454.819,A -85,B 0,C 180,E1 -2874.953,E2 -2874.953} C_VEL
LIN {X 0,Y 559.243,Z 454.819,A -85,B 0,C 180,E1 -2877.839,E2 -2877.839} C_VEL
LIN {X 0,Y 559.268,Z 454.814,A -85,B 0,C 180,E1 -2880.72,E2 -2880.72} C_VEL
LIN {X 0,Y 559.237,Z 454.819,A -85,B 0,C 180,E1 -2882.881,E2 -2882.881} C_VEL
LIN {X 0,Y 559.221,Z 454.825,A -85,B 0,C 180,E1 -2885.77,E2 -2885.77} C_VEL
LIN {X 0,Y 559.194,Z 454.823,A -85,B 0,C 180,E1 -2888.674,E2 -2888.674} C_VEL
LIN {X 0,Y 559.199,Z 454.831,A -85,B 0,C 180,E1 -2891.601,E2 -2891.601} C_VEL
LIN {X 0,Y 559.189,Z 454.824,A -85,B 0,C 180,E1 -2894.596,E2 -2894.596} C_VEL
LIN {X 0,Y 559.155,Z 454.834,A -85,B 0,C 180,E1 -2897.557,E2 -2897.557} C_VEL
LIN {X 0,Y 559.166,Z 454.831,A -85,B 0,C 180,E1 -2899.838,E2 -2899.838} C_VEL
LIN {X 0,Y 559.134,Z 454.833,A -85,B 0,C 180,E1 -2902.153,E2 -2902.153} C_VEL
LIN {X 0,Y 559.171,Z 454.829,A -85,B 0,C 180,E1 -2905.188,E2 -2905.188} C_VEL
LIN {X 0,Y 559.187,Z 454.832,A -85,B 0,C 180,E1 -2907.712,E2 -2907.712} C_VEL
LIN {X 0,Y 559.161,Z 454.83,A -85,B 0,C 180,E1 -2910.182,E2 -2910.182} C_VEL
LIN {X 0,Y 559.168,Z 454.824,A -85,B 0,C 180,E1 -2912.715,E2 -2912.715} C_VEL
LIN {X 0,Y 559.152,Z 454.832,A -85,B 0,C 180,E1 -2915.322,E2 -2915.322} C_VEL
LIN {X 0,Y 559.129,Z 454.836,A -85,B 0,C 180,E1 -2918.018,E2 -2918.018} C_VEL
LIN {X 0,Y 559.171,Z 454.827,A -85,B 0,C 180,E1 -2920.811,E2 -2920.811} C_VEL
LIN {X 0,Y 559.136,Z 454.834,A -85,B 0,C 180,E1 -2923.735,E2 -2923.735} C_VEL
LIN {X 0,Y 559.164,Z 454.828,A -85,B 0,C 180,E1 -2926.802,E2 -2926.802} C_VEL
LIN {X 0,Y 559.173,Z 454.826,A -85,B 0,C 180,E1 -2929.19,E2 -2929.19} C_VEL
LIN {X 0,Y 559.133,Z 454.839,A -85,B 0,C 180,E1 -2931.984,E2 -2931.984} C_VEL
LIN {X 0,Y 559.143,Z 454.831,A -85,B 0,C 180,E1 -2934.786,E2 -2934.786} C_VEL
LIN {X 0,Y 559.156,Z 454.831,A -85,B 0,C 180,E1 -2937.365,E2 -2937.365} C_VEL
LIN {X 0,Y 559.149,Z 454.826,A -85,B 0,C 180,E1 -2940.143,E2 -2940.143} C_VEL
LIN {X 0,Y 559.226,Z 455,A -85,B 0,C 180,E1 -2942.382,E2 -2942.382} C_VEL
LIN {X 0,Y 561.049,Z 463.12,A -85,B 0,C 180,E1 -2943.397,E2 -2943.397} C_VEL
LIN {X 0,Y 560.897,Z 484.303,A -85,B 0,C 180,E1 -2945.773,E2 -2945.773} C_VEL
LIN {X 0,Y 560.582,Z 507.862,A -85,B 0,C 180,E1 -2948.402,E2 -2948.402} C_VEL
LIN {X 0,Y 560.117,Z 533.822,A -85,B 0,C 180,E1 -2951.34,E2 -2951.34} C_VEL
LIN {X 0,Y 559.749,Z 559.037,A -85,B 0,C 180,E1 -2954.152,E2 -2954.152} C_VEL
LIN {X 0,Y 559.602,Z 573.904,A -85,B 0,C 180,E1 -2955.778,E2 -2955.778} C_VEL
LIN {X 0,Y 560.328,Z 581.535,A -85,B 0,C 180,E1 -2955.913,E2 -2955.913} C_VEL
LIN {X 0,Y 560.068,Z 683.962,A -85,B 0,C 180,E1 -2957.246,E2 -2957.246} C_VEL
LIN {X 0,Y 559.971,Z 696.466,A -85,B 0,C 180,E1 -2957.543,E2 -2957.543} C_VEL
LIN {X 0,Y 559.79,Z 708.926,A -85,B 0,C 180,E1 -2957.98,E2 -2957.98} C_VEL
LIN {X 0,Y 559.668,Z 720.814,A -85,B 0,C 180,E1 -2958.547,E2 -2958.547} C_VEL
LIN {X 0,Y 559.507,Z 731.912,A -85,B 0,C 180,E1 -2959.232,E2 -2959.232} C_VEL
LIN {X 0,Y 559.309,Z 742.543,A -85,B 0,C 180,E1 -2960.051,E2 -2960.051} C_VEL
LIN {X 0,Y 559.161,Z 752.115,A -85,B 0,C 180,E1 -2960.961,E2 -2960.961} C_VEL
LIN {X 0,Y 559.05,Z 759.962,A -85,B 0,C 180,E1 -2961.87,E2 -2961.87} C_VEL
LIN {X 0,Y 558.944,Z 767.623,A -85,B 0,C 180,E1 -2962.959,E2 -2962.959} C_VEL
LIN {X 0,Y 558.935,Z 774.68,A -85,B 0,C 180,E1 -2964.227,E2 -2964.227} C_VEL
LIN {X 0,Y 558.827,Z 779.373,A -85,B 0,C 180,E1 -2965.311,E2 -2965.311} C_VEL
LIN {X 0,Y 558.836,Z 782.958,A -85,B 0,C 180,E1 -2966.395,E2 -2966.395} C_VEL
LIN {X 0,Y 558.799,Z 784.808,A -85,B 0,C 180,E1 -2967.116,E2 -2967.116} C_VEL
LIN {X 0,Y 558.745,Z 787.185,A -85,B 0,C 180,E1 -2968.559,E2 -2968.559} C_VEL
LIN {X 0,Y 558.74,Z 788,A -85,B 0,C 180,E1 -2970,E2 -2970} C_VEL
LIN {X 0,Y 558.745,Z 787.186,A -85,B 0,C 180,E1 -2971.441,E2 -2971.441} C_VEL
LIN {X 0,Y 558.799,Z 784.81,A -85,B 0,C 180,E1 -2972.884,E2 -2972.884} C_VEL
LIN {X 0,Y 558.843,Z 781.896,A -85,B 0,C 180,E1 -2973.966,E2 -2973.966} C_VEL
LIN {X 0,Y 558.799,Z 777.949,A -85,B 0,C 180,E1 -2975.051,E2 -2975.051} C_VEL
LIN {X 0,Y 558.921,Z 772.868,A -85,B 0,C 180,E1 -2976.135,E2 -2976.135} C_VEL
LIN {X 0,Y 558.977,Z 766.469,A -85,B 0,C 180,E1 -2977.223,E2 -2977.223} C_VEL
LIN {X 0,Y 559.099,Z 758.48,A -85,B 0,C 180,E1 -2978.311,E2 -2978.311} C_VEL
LIN {X 0,Y 559.184,Z 750.337,A -85,B 0,C 180,E1 -2979.221,E2 -2979.221} C_VEL
LIN {X 0,Y 559.339,Z 740.403,A -85,B 0,C 180,E1 -2980.131,E2 -2980.131} C_VEL
LIN {X 0,Y 559.53,Z 729.368,A -85,B 0,C 180,E1 -2980.939,E2 -2980.939} C_VEL
LIN {X 0,Y 559.703,Z 717.148,A -85,B 0,C 180,E1 -2981.643,E2 -2981.643} C_VEL
LIN {X 0,Y 559.822,Z 704.776,A -85,B 0,C 180,E1 -2982.184,E2 -2982.184} C_VEL
LIN {X 0,Y 559.962,Z 692.274,A -85,B 0,C 180,E1 -2982.572,E2 -2982.572} C_VEL
LIN {X 0,Y 560.089,Z 679.622,A -85,B 0,C 180,E1 -2982.823,E2 -2982.823} C_VEL
LIN {X 0,Y 560.195,Z 578.629,A -85,B 0,C 180,E1 -2984.128,E2 -2984.128} C_VEL
LIN {X 0,Y 559.602,Z 573.905,A -85,B 0,C 180,E1 -2984.222,E2 -2984.222} C_VEL
LIN {X 0,Y 559.907,Z 546.759,A -85,B 0,C 180,E1 -2987.213,E2 -2987.213} C_VEL
LIN {X 0,Y 560.392,Z 518.695,A -85,B 0,C 180,E1 -2990.365,E2 -2990.365} C_VEL
LIN {X 0,Y 560.805,Z 494.916,A -85,B 0,C 180,E1 -2993.055,E2 -2993.055} C_VEL
LIN {X 0,Y 561.093,Z 466.643,A -85,B 0,C 180,E1 -2996.201,E2 -2996.201} C_VEL
LIN {X 0,Y 561.059,Z 463.094,A -85,B 0,C 180,E1 -2996.603,E2 -2996.603} C_VEL
LIN {X 0,Y 559.197,Z 454.926,A -85,B 0,C 180,E1 -2997.64,E2 -2997.64} C_VEL
LIN {X 0,Y 559.156,Z 454.827,A -85,B 0,C 180,E1 -3000.182,E2 -3000.182} C_VEL
LIN {X 0,Y 559.156,Z 454.83,A -85,B 0,C 180,E1 -3002.714,E2 -3002.714} C_VEL
LIN {X 0,Y 559.125,Z 454.834,A -85,B 0,C 180,E1 -3005.323,E2 -3005.323} C_VEL
LIN {X 0,Y 559.133,Z 454.838,A -85,B 0,C 180,E1 -3008.017,E2 -3008.017} C_VEL
LIN {X 0,Y 559.173,Z 454.826,A -85,B 0,C 180,E1 -3010.81,E2 -3010.81} C_VEL
LIN {X 0,Y 559.159,Z 454.831,A -85,B 0,C 180,E1 -3013.731,E2 -3013.731} C_VEL
LIN {X 0,Y 559.141,Z 454.829,A -85,B 0,C 180,E1 -3016.803,E2 -3016.803} C_VEL
LIN {X 0,Y 559.171,Z 454.827,A -85,B 0,C 180,E1 -3019.189,E2 -3019.189} C_VEL
LIN {X 0,Y 559.129,Z 454.835,A -85,B 0,C 180,E1 -3021.982,E2 -3021.982} C_VEL
LIN {X 0,Y 559.154,Z 454.831,A -85,B 0,C 180,E1 -3024.782,E2 -3024.782} C_VEL
LIN {X 0,Y 559.167,Z 454.825,A -85,B 0,C 180,E1 -3027.361,E2 -3027.361} C_VEL
LIN {X 0,Y 559.182,Z 454.832,A -85,B 0,C 180,E1 -3030.134,E2 -3030.134} C_VEL
LIN {X 0,Y 559.174,Z 454.822,A -85,B 0,C 180,E1 -3033.169,E2 -3033.169} C_VEL
LIN {X 0,Y 559.148,Z 454.829,A -85,B 0,C 180,E1 -3035.494,E2 -3035.494} C_VEL
LIN {X 0,Y 559.168,Z 454.831,A -85,B 0,C 180,E1 -3038.624,E2 -3038.624} C_VEL
LIN {X 0,Y 559.163,Z 454.825,A -85,B 0,C 180,E1 -3040.926,E2 -3040.926} C_VEL
LIN {X 0,Y 559.162,Z 454.829,A -85,B 0,C 180,E1 -3043.948,E2 -3043.948} C_VEL
LIN {X 0,Y 559.165,Z 454.832,A -85,B 0,C 180,E1 -3046.184,E2 -3046.184} C_VEL
LIN {X 0,Y 559.201,Z 454.822,A -85,B 0,C 180,E1 -3049.134,E2 -3049.134} C_VEL
LIN {X 0,Y 559.204,Z 454.825,A -85,B 0,C 180,E1 -3052.054,E2 -3052.054} C_VEL
LIN {X 0,Y 559.252,Z 454.817,A -85,B 0,C 180,E1 -3054.953,E2 -3054.953} C_VEL
LIN {X 0,Y 559.243,Z 454.817,A -85,B 0,C 180,E1 -3057.839,E2 -3057.839} C_VEL
LIN {X 0,Y 559.269,Z 454.821,A -85,B 0,C 180,E1 -3060.72,E2 -3060.72} C_VEL
LIN {X 0,Y 559.237,Z 454.822,A -85,B 0,C 180,E1 -3062.881,E2 -3062.881} C_VEL
LIN {X 0,Y 559.227,Z 454.819,A -85,B 0,C 180,E1 -3065.77,E2 -3065.77} C_VEL
LIN {X 0,Y 559.195,Z 454.83,A -85,B 0,C 180,E1 -3068.674,E2 -3068.674} C_VEL
LIN {X 0,Y 559.199,Z 454.822,A -85,B 0,C 180,E1 -3071.601,E2 -3071.601} C_VEL
LIN {X 0,Y 559.189,Z 454.832,A -85,B 0,C 180,E1 -3074.596,E2 -3074.596} C_VEL
LIN {X 0,Y 559.155,Z 454.828,A -85,B 0,C 180,E1 -3077.557,E2 -3077.557} C_VEL
LIN {X 0,Y 559.166,Z 454.827,A -85,B 0,C 180,E1 -3079.838,E2 -3079.838} C_VEL
LIN {X 0,Y 559.135,Z 454.831,A -85,B 0,C 180,E1 -3082.153,E2 -3082.153} C_VEL
LIN {X 0,Y 559.171,Z 454.83,A -85,B 0,C 180,E1 -3085.188,E2 -3085.188} C_VEL
LIN {X 0,Y 559.187,Z 454.822,A -85,B 0,C 180,E1 -3087.712,E2 -3087.712} C_VEL
LIN {X 0,Y 559.146,Z 454.826,A -85,B 0,C 180,E1 -3090.634,E2 -3090.634} C_VEL
LIN {X 0,Y 558.484,Z 454.914,A -85,B 0,C 180,E1 -3091.235,E2 -3091.235} C_VEL
LIN {X 0,Y 555.621,Z 455.271,A -85,B 0,C 180,E1 -3092.211,E2 -3092.211} C_VEL
LIN {X 0,Y 553.209,Z 455.576,A -85,B 0,C 180,E1 -3092.997,E2 -3092.997} C_VEL
LIN {X 0,Y 552.191,Z 455.696,A -85,B 0,C 180,E1 -3093.604,E2 -3093.604} C_VEL
LIN {X 0,Y 552.118,Z 455.704,A -85,B 0,C 180,E1 -3093.809,E2 -3093.809} C_VEL
LIN {X 0,Y 552.106,Z 455.714,A -85,B 0,C 180,E1 -3096.747,E2 -3096.747} C_VEL
LIN {X 0,Y 552.13,Z 455.698,A -85,B 0,C 180,E1 -3099.527,E2 -3099.527} C_VEL
LIN {X 0,Y 552.126,Z 455.705,A -85,B 0,C 180,E1 -3102.426,E2 -3102.426} C_VEL
LIN {X 0,Y 552.096,Z 455.708,A -85,B 0,C 180,E1 -3105.564,E2 -3105.564} C_VEL
LIN {X 0,Y 552.138,Z 455.704,A -85,B 0,C 180,E1 -3108.677,E2 -3108.677} C_VEL
LIN {X 0,Y 552.119,Z 455.708,A -85,B 0,C 180,E1 -3111.412,E2 -3111.412} C_VEL
LIN {X 0,Y 552.101,Z 455.7,A -85,B 0,C 180,E1 -3114.159,E2 -3114.159} C_VEL
LIN {X 0,Y 552.122,Z 455.7,A -85,B 0,C 180,E1 -3116.816,E2 -3116.816} C_VEL
LIN {X 0,Y 552.108,Z 455.712,A -85,B 0,C 180,E1 -3119.392,E2 -3119.392} C_VEL
LIN {X 0,Y 552.11,Z 455.702,A -85,B 0,C 180,E1 -3121.902,E2 -3121.902} C_VEL
LIN {X 0,Y 552.157,Z 455.701,A -85,B 0,C 180,E1 -3124.65,E2 -3124.65} C_VEL
LIN {X 0,Y 552.095,Z 455.708,A -85,B 0,C 180,E1 -3127.55,E2 -3127.55} C_VEL
LIN {X 0,Y 552.151,Z 455.703,A -85,B 0,C 180,E1 -3130.374,E2 -3130.374} C_VEL
LIN {X 0,Y 552.137,Z 455.691,A -85,B 0,C 180,E1 -3132.977,E2 -3132.977} C_VEL
LIN {X 0,Y 552.208,Z 455.903,A -85,B 0,C 180,E1 -3135.944,E2 -3135.944} C_VEL
LIN {X 0,Y 552.466,Z 457.024,A -85,B 0,C 180,E1 -3136.06,E2 -3136.06} C_VEL
LIN {X 0,Y 553.428,Z 460.01,A -85,B 0,C 180,E1 -3136.132,E2 -3136.132} C_VEL
LIN {X 0,Y 553.207,Z 535.279,A -85,B 0,C 180,E1 -3137.132,E2 -3137.132} C_VEL
LIN {X 0,Y 553.089,Z 548.458,A -85,B 0,C 180,E1 -3137.455,E2 -3137.455} C_VEL
LIN {X 0,Y 552.917,Z 560.518,A -85,B 0,C 180,E1 -3137.894,E2 -3137.894} C_VEL
LIN {X 0,Y 552.762,Z 571.896,A -85,B 0,C 180,E1 -3138.452,E2 -3138.452} C_VEL
LIN {X 0,Y 552.581,Z 583.412,A -85,B 0,C 180,E1 -3139.188,E2 -3139.188} C_VEL
LIN {X 0,Y 552.364,Z 593.773,A -85,B 0,C 180,E1 -3140.017,E2 -3140.017} C_VEL
LIN {X 0,Y 552.198,Z 602.222,A -85,B 0,C 180,E1 -3140.846,E2 -3140.846} C_VEL
LIN {X 0,Y 552.037,Z 609.989,A -85,B 0,C 180,E1 -3141.766,E2 -3141.766} C_VEL
LIN {X 0,Y 551.917,Z 617.675,A -85,B 0,C 180,E1 -3142.887,E2 -3142.887} C_VEL
LIN {X 0,Y 551.868,Z 624.508,A -85,B 0,C 180,E1 -3144.153,E2 -3144.153} C_VEL
LIN {X 0,Y 551.725,Z 629.201,A -85,B 0,C 180,E1 -3145.251,E2 -3145.251} C_VEL
LIN {X 0,Y 551.75,Z 632.829,A -85,B 0,C 180,E1 -3146.349,E2 -3146.349} C_VEL
LIN {X 0,Y 551.723,Z 634.708,A -85,B 0,C 180,E1 -3147.079,E2 -3147.079} C_VEL
LIN {X 0,Y 551.656,Z 636.128,A -85,B 0,C 180,E1 -3147.81,E2 -3147.81} C_VEL
LIN {X 0,Y 551.642,Z 637.756,A -85,B 0,C 180,E1 -3149.27,E2 -3149.27} C_VEL
LIN {X 0,Y 551.641,Z 637.996,A -85,B 0,C 180,E1 -3150,E2 -3150} C_VEL
LIN {X 0,Y 551.641,Z 637.815,A -85,B 0,C 180,E1 -3150.73,E2 -3150.73} C_VEL
LIN {X 0,Y 551.657,Z 636.266,A -85,B 0,C 180,E1 -3152.19,E2 -3152.19} C_VEL
LIN {X 0,Y 551.724,Z 634.905,A -85,B 0,C 180,E1 -3152.921,E2 -3152.921} C_VEL
LIN {X 0,Y 551.764,Z 632.025,A -85,B 0,C 180,E1 -3154.017,E2 -3154.017} C_VEL
LIN {X 0,Y 551.723,Z 628.128,A -85,B 0,C 180,E1 -3155.116,E2 -3155.116} C_VEL
LIN {X 0,Y 551.833,Z 622.496,A -85,B 0,C 180,E1 -3156.349,E2 -3156.349} C_VEL
LIN {X 0,Y 551.925,Z 615.799,A -85,B 0,C 180,E1 -3157.499,E2 -3157.499} C_VEL
LIN {X 0,Y 552.113,Z 607.782,A -85,B 0,C 180,E1 -3158.602,E2 -3158.602} C_VEL
LIN {X 0,Y 552.255,Z 599.573,A -85,B 0,C 180,E1 -3159.522,E2 -3159.522} C_VEL
LIN {X 0,Y 552.482,Z 589.416,A -85,B 0,C 180,E1 -3160.444,E2 -3160.444} C_VEL
LIN {X 0,Y 552.696,Z 578.841,A -85,B 0,C 180,E1 -3161.214,E2 -3161.214} C_VEL
LIN {X 0,Y 552.819,Z 568.467,A -85,B 0,C 180,E1 -3161.82,E2 -3161.82} C_VEL
LIN {X 0,Y 552.962,Z 557.079,A -85,B 0,C 180,E1 -3162.338,E2 -3162.338} C_VEL
LIN {X 0,Y 553.107,Z 544.336,A -85,B 0,C 180,E1 -3162.754,E2 -3162.754} C_VEL
LIN {X 0,Y 553.235,Z 532.256,A -85,B 0,C 180,E1 -3163.008,E2 -3163.008} C_VEL
LIN {X 0,Y 553.276,Z 459.494,A -85,B 0,C 180,E1 -3163.969,E2 -3163.969} C_VEL
LIN {X 0,Y 552.359,Z 456.639,A -85,B 0,C 180,E1 -3164.052,E2 -3164.052} C_VEL
LIN {X 0,Y 552.17,Z 455.747,A -85,B 0,C 180,E1 -3164.202,E2 -3164.202} C_VEL
LIN {X 0,Y 552.138,Z 455.691,A -85,B 0,C 180,E1 -3167.32,E2 -3167.32} C_VEL
LIN {X 0,Y 552.133,Z 455.705,A -85,B 0,C 180,E1 -3170.101,E2 -3170.101} C_VEL
LIN {X 0,Y 552.094,Z 455.708,A -85,B 0,C 180,E1 -3172.45,E2 -3172.45} C_VEL
LIN {X 0,Y 552.157,Z 455.703,A -85,B 0,C 180,E1 -3175.35,E2 -3175.35} C_VEL
LIN {X 0,Y 552.11,Z 455.701,A -85,B 0,C 180,E1 -3178.098,E2 -3178.098} C_VEL
LIN {X 0,Y 552.108,Z 455.711,A -85,B 0,C 180,E1 -3180.608,E2 -3180.608} C_VEL
LIN {X 0,Y 552.12,Z 455.712,A -85,B 0,C 180,E1 -3183.185,E2 -3183.185} C_VEL
LIN {X 0,Y 552.1,Z 455.706,A -85,B 0,C 180,E1 -3185.842,E2 -3185.842} C_VEL
LIN {X 0,Y 552.124,Z 455.714,A -85,B 0,C 180,E1 -3189.061,E2 -3189.061} C_VEL
LIN {X 0,Y 552.137,Z 455.704,A -85,B 0,C 180,E1 -3191.443,E2 -3191.443} C_VEL
LIN {X 0,Y 552.093,Z 455.709,A -85,B 0,C 180,E1 -3194.531,E2 -3194.531} C_VEL
LIN {X 0,Y 552.126,Z 455.706,A -85,B 0,C 180,E1 -3197.584,E2 -3197.584} C_VEL
LIN {X 0,Y 552.13,Z 455.697,A -85,B 0,C 180,E1 -3200.473,E2 -3200.473} C_VEL
LIN {X 0,Y 552.109,Z 455.714,A -85,B 0,C 180,E1 -3203.315,E2 -3203.315} C_VEL
LIN {X 0,Y 552.134,Z 455.702,A -85,B 0,C 180,E1 -3205.939,E2 -3205.939} C_VEL
LIN {X 0,Y 552.111,Z 455.701,A -85,B 0,C 180,E1 -3208.54,E2 -3208.54} C_VEL
LIN {X 0,Y 552.12,Z 455.709,A -85,B 0,C 180,E1 -3211.436,E2 -3211.436} C_VEL
LIN {X 0,Y 552.13,Z 455.704,A -85,B 0,C 180,E1 -3214.356,E2 -3214.356} C_VEL
LIN {X 0,Y 552.102,Z 455.709,A -85,B 0,C 180,E1 -3216.758,E2 -3216.758} C_VEL
LIN {X 0,Y 552.118,Z 455.71,A -85,B 0,C 180,E1 -3219.12,E2 -3219.12} C_VEL
LIN {X 0,Y 552.123,Z 455.711,A -85,B 0,C 180,E1 -3221.444,E2 -3221.444} C_VEL
LIN {X 0,Y 552.111,Z 455.707,A -85,B 0,C 180,E1 -3223.737,E2 -3223.737} C_VEL
LIN {X 0,Y 552.127,Z 455.705,A -85,B 0,C 180,E1 -3226.004,E2 -3226.004} C_VEL
LIN {X 0,Y 552.169,Z 455.702,A -85,B 0,C 180,E1 -3228.993,E2 -3228.993} C_VEL
LIN {X 0,Y 552.155,Z 455.701,A -85,B 0,C 180,E1 -3231.951,E2 -3231.951} C_VEL
LIN {X 0,Y 552.226,Z 455.693,A -85,B 0,C 180,E1 -3234.889,E2 -3234.889} C_VEL
LIN {X 0,Y 552.214,Z 455.695,A -85,B 0,C 180,E1 -3237.812,E2 -3237.812} C_VEL
LIN {X 0,Y 552.238,Z 455.69,A -85,B 0,C 180,E1 -3240.729,E2 -3240.729} C_VEL
LIN {X 0,Y 552.203,Z 455.695,A -85,B 0,C 180,E1 -3242.918,E2 -3242.918} C_VEL
LIN {X 0,Y 552.191,Z 455.7,A -85,B 0,C 180,E1 -3245.844,E2 -3245.844} C_VEL
LIN {X 0,Y 552.162,Z 455.7,A -85,B 0,C 180,E1 -3248.786,E2 -3248.786} C_VEL
LIN {X 0,Y 552.155,Z 455.706,A -85,B 0,C 180,E1 -3251.751,E2 -3251.751} C_VEL
LIN {X 0,Y 552.126,Z 455.704,A -85,B 0,C 180,E1 -3254.749,E2 -3254.749} C_VEL
LIN {X 0,Y 552.106,Z 455.707,A -85,B 0,C 180,E1 -3257.789,E2 -3257.789} C_VEL
LIN {X 0,Y 552.125,Z 455.704,A -85,B 0,C 180,E1 -3260.101,E2 -3260.101} C_VEL
LIN {X 0,Y 552.087,Z 455.709,A -85,B 0,C 180,E1 -3262.451,E2 -3262.451} C_VEL
LIN {X 0,Y 552.148,Z 455.706,A -85,B 0,C 180,E1 -3265.351,E2 -3265.351} C_VEL
LIN {X 0,Y 552.119,Z 455.707,A -85,B 0,C 180,E1 -3268.098,E2 -3268.098} C_VEL
LIN {X 0,Y 552.106,Z 455.707,A -85,B 0,C 180,E1 -3270.609,E2 -3270.609} C_VEL
LIN {X 0,Y 552.122,Z 455.704,A -85,B 0,C 180,E1 -3273.185,E2 -3273.185} C_VEL
LIN {X 0,Y 552.107,Z 455.714,A -85,B 0,C 180,E1 -3275.842,E2 -3275.842} C_VEL
LIN {X 0,Y 552.12,Z 455.705,A -85,B 0,C 180,E1 -3279.063,E2 -3279.063} C_VEL
LIN {X 0,Y 552.134,Z 455.708,A -85,B 0,C 180,E1 -3281.445,E2 -3281.445} C_VEL
LIN {X 0,Y 552.09,Z 455.705,A -85,B 0,C 180,E1 -3284.533,E2 -3284.533} C_VEL
LIN {X 0,Y 552.127,Z 455.711,A -85,B 0,C 180,E1 -3287.585,E2 -3287.585} C_VEL
LIN {X 0,Y 552.131,Z 455.705,A -85,B 0,C 180,E1 -3290.474,E2 -3290.474} C_VEL
LIN {X 0,Y 552.109,Z 455.708,A -85,B 0,C 180,E1 -3293.317,E2 -3293.317} C_VEL
LIN {X 0,Y 552.126,Z 455.711,A -85,B 0,C 180,E1 -3295.94,E2 -3295.94} C_VEL
LIN {X 0,Y 552.118,Z 455.706,A -85,B 0,C 180,E1 -3298.541,E2 -3298.541} C_VEL
LIN {X 0,Y 552.124,Z 455.711,A -85,B 0,C 180,E1 -3301.439,E2 -3301.439} C_VEL
LIN {X 0,Y 552.189,Z 455.935,A -85,B 0,C 180,E1 -3302.216,E2 -3302.216} C_VEL
LIN {X 0,Y 554.219,Z 465.799,A -85,B 0,C 180,E1 -3303.449,E2 -3303.449} C_VEL
LIN {X 0,Y 553.858,Z 492.268,A -85,B 0,C 180,E1 -3306.441,E2 -3306.441} C_VEL
LIN {X 0,Y 553.536,Z 518.659,A -85,B 0,C 180,E1 -3309.371,E2 -3309.371} C_VEL
LIN {X 0,Y 553.011,Z 546.389,A -85,B 0,C 180,E1 -3312.524,E2 -3312.524} C_VEL
LIN {X 0,Y 552.647,Z 573.908,A -85,B 0,C 180,E1 -3315.595,E2 -3315.595} C_VEL
LIN {X 0,Y 553.452,Z 581.535,A -85,B 0,C 180,E1 -3315.734,E2 -3315.734} C_VEL
LIN {X 0,Y 553.167,Z 683.962,A -85,B 0,C 180,E1 -3317.084,E2 -3317.084} C_VEL
LIN {X 0,Y 553.022,Z 696.466,A -85,B 0,C 180,E1 -3317.384,E2 -3317.384} C_VEL
LIN {X 0,Y 552.849,Z 709.376,A -85,B 0,C 180,E1 -3317.846,E2 -3317.846} C_VEL
LIN {X 0,Y 552.689,Z 721.675,A -85,B 0,C 180,E1 -3318.45,E2 -3318.45} C_VEL
LIN {X 0,Y 552.505,Z 733.201,A -85,B 0,C 180,E1 -3319.186,E2 -3319.186} C_VEL
LIN {X 0,Y 552.295,Z 743.606,A -85,B 0,C 180,E1 -3320.016,E2 -3320.016} C_VEL
LIN {X 0,Y 552.125,Z 752.115,A -85,B 0,C 180,E1 -3320.845,E2 -3320.845} C_VEL
LIN {X 0,Y 552.013,Z 759.962,A -85,B 0,C 180,E1 -3321.765,E2 -3321.765} C_VEL
LIN {X 0,Y 551.889,Z 767.622,A -85,B 0,C 180,E1 -3322.868,E2 -3322.868} C_VEL
LIN {X 0,Y 551.867,Z 774.68,A -85,B 0,C 180,E1 -3324.153,E2 -3324.153} C_VEL
LIN {X 0,Y 551.725,Z 779.373,A -85,B 0,C 180,E1 -3325.251,E2 -3325.251} C_VEL
LIN {X 0,Y 551.75,Z 782.958,A -85,B 0,C 180,E1 -3326.349,E2 -3326.349} C_VEL
LIN {X 0,Y 551.724,Z 784.808,A -85,B 0,C 180,E1 -3327.079,E2 -3327.079} C_VEL
LIN {X 0,Y 551.645,Z 787.184,A -85,B 0,C 180,E1 -3328.54,E2 -3328.54} C_VEL
LIN {X 0,Y 551.64,Z 788,A -85,B 0,C 180,E1 -3330,E2 -3330} C_VEL
LIN {X 0,Y 551.645,Z 787.185,A -85,B 0,C 180,E1 -3331.46,E2 -3331.46} C_VEL
LIN {X 0,Y 551.724,Z 784.81,A -85,B 0,C 180,E1 -3332.921,E2 -3332.921} C_VEL
LIN {X 0,Y 551.763,Z 781.896,A -85,B 0,C 180,E1 -3334.017,E2 -3334.017} C_VEL
LIN {X 0,Y 551.724,Z 777.949,A -85,B 0,C 180,E1 -3335.116,E2 -3335.116} C_VEL
LIN {X 0,Y 551.803,Z 772.19,A -85,B 0,C 180,E1 -3336.341,E2 -3336.341} C_VEL
LIN {X 0,Y 551.926,Z 765.238,A -85,B 0,C 180,E1 -3337.499,E2 -3337.499} C_VEL
LIN {X 0,Y 552.082,Z 756.993,A -85,B 0,C 180,E1 -3338.602,E2 -3338.602} C_VEL
LIN {X 0,Y 552.222,Z 748.541,A -85,B 0,C 180,E1 -3339.523,E2 -3339.523} C_VEL
LIN {X 0,Y 552.384,Z 738.098,A -85,B 0,C 180,E1 -3340.445,E2 -3340.445} C_VEL
LIN {X 0,Y 552.622,Z 727.134,A -85,B 0,C 180,E1 -3341.223,E2 -3341.223} C_VEL
LIN {X 0,Y 552.781,Z 716.413,A -85,B 0,C 180,E1 -3341.83,E2 -3341.83} C_VEL
LIN {X 0,Y 552.882,Z 704.772,A -85,B 0,C 180,E1 -3342.34,E2 -3342.34} C_VEL
LIN {X 0,Y 553.017,Z 692.273,A -85,B 0,C 180,E1 -3342.733,E2 -3342.733} C_VEL
LIN {X 0,Y 553.178,Z 679.621,A -85,B 0,C 180,E1 -3342.986,E2 -3342.986} C_VEL
LIN {X 0,Y 553.38,Z 579.746,A -85,B 0,C 180,E1 -3344.291,E2 -3344.291} C_VEL
LIN {X 0,Y 552.65,Z 573.911,A -85,B 0,C 180,E1 -3344.405,E2 -3344.405} C_VEL
LIN {X 0,Y 553.011,Z 546.389,A -85,B 0,C 180,E1 -3347.476,E2 -3347.476} C_VEL
LIN {X 0,Y 553.536,Z 518.659,A -85,B 0,C 180,E1 -3350.629,E2 -3350.629} C_VEL
LIN {X 0,Y 553.896,Z 490.507,A -85,B 0,C 180,E1 -3353.756,E2 -3353.756} C_VEL
LIN {X 0,Y 554.226,Z 465.783,A -85,B 0,C 180,E1 -3356.55,E2 -3356.55} C_VEL
LIN {X 0,Y 552.193,Z 455.828,A -85,B 0,C 180,E1 -3357.809,E2 -3357.809} C_VEL
LIN {X 0,Y 552.107,Z 455.708,A -85,B 0,C 180,E1 -3360.608,E2 -3360.608} C_VEL
LIN {X 0,Y 552.114,Z 455.705,A -85,B 0,C 180,E1 -3363.185,E2 -3363.185} C_VEL
LIN {X 0,Y 552.083,Z 455.716,A -85,B 0,C 180,E1 -3365.843,E2 -3365.843} C_VEL
LIN {X 0,Y 552.123,Z 455.704,A -85,B 0,C 180,E1 -3369.061,E2 -3369.061} C_VEL
LIN {X 0,Y 552.137,Z 455.702,A -85,B 0,C 180,E1 -3371.443,E2 -3371.443} C_VEL
LIN {X 0,Y 552.092,Z 455.709,A -85,B 0,C 180,E1 -3374.531,E2 -3374.531} C_VEL
LIN {X 0,Y 552.126,Z 455.702,A -85,B 0,C 180,E1 -3377.584,E2 -3377.584} C_VEL
LIN {X 0,Y 552.129,Z 455.709,A -85,B 0,C 180,E1 -3380.473,E2 -3380.473} C_VEL
LIN {X 0,Y 552.108,Z 455.706,A -85,B 0,C 180,E1 -3383.315,E2 -3383.315} C_VEL
LIN {X 0,Y 552.134,Z 455.707,A -85,B 0,C 180,E1 -3385.939,E2 -3385.939} C_VEL
LIN {X 0,Y 552.111,Z 455.713,A -85,B 0,C 180,E1 -3388.54,E2 -3388.54} C_VEL
LIN {X 0,Y 552.119,Z 455.704,A -85,B 0,C 180,E1 -3391.437,E2 -3391.437} C_VEL
LIN {X 0,Y 552.129,Z 455.709,A -85,B 0,C 180,E1 -3394.356,E2 -3394.356} C_VEL
LIN {X 0,Y 552.101,Z 455.711,A -85,B 0,C 180,E1 -3396.758,E2 -3396.758} C_VEL
LIN {X 0,Y 552.118,Z 455.703,A -85,B 0,C 180,E1 -3399.12,E2 -3399.12} C_VEL
LIN {X 0,Y 552.122,Z 455.698,A -85,B 0,C 180,E1 -3401.444,E2 -3401.444} C_VEL
LIN {X 0,Y 552.112,Z 455.705,A -85,B 0,C 180,E1 -3403.737,E2 -3403.737} C_VEL
LIN {X 0,Y 552.127,Z 455.707,A -85,B 0,C 180,E1 -3406.004,E2 -3406.004} C_VEL
LIN {X 0,Y 552.169,Z 455.699,A -85,B 0,C 180,E1 -3408.994,E2 -3408.994} C_VEL
LIN {X 0,Y 552.157,Z 455.702,A -85,B 0,C 180,E1 -3411.952,E2 -3411.952} C_VEL
LIN {X 0,Y 552.226,Z 455.693,A -85,B 0,C 180,E1 -3414.889,E2 -3414.889} C_VEL
LIN {X 0,Y 552.215,Z 455.693,A -85,B 0,C 180,E1 -3417.812,E2 -3417.812} C_VEL
LIN {X 0,Y 552.239,Z 455.696,A -85,B 0,C 180,E1 -3420.729,E2 -3420.729} C_VEL
LIN {X 0,Y 552.203,Z 455.697,A -85,B 0,C 180,E1 -3422.918,E2 -3422.918} C_VEL
LIN {X 0,Y 552.198,Z 455.695,A -85,B 0,C 180,E1 -3425.844,E2 -3425.844} C_VEL
LIN {X 0,Y 552.163,Z 455.704,A -85,B 0,C 180,E1 -3428.786,E2 -3428.786} C_VEL
LIN {X 0,Y 552.155,Z 455.7,A -85,B 0,C 180,E1 -3431.751,E2 -3431.751} C_VEL
LIN {X 0,Y 552.127,Z 455.711,A -85,B 0,C 180,E1 -3434.749,E2 -3434.749} C_VEL
LIN {X 0,Y 552.107,Z 455.706,A -85,B 0,C 180,E1 -3437.789,E2 -3437.789} C_VEL
LIN {X 0,Y 552.126,Z 455.705,A -85,B 0,C 180,E1 -3440.102,E2 -3440.102} C_VEL
LIN {X 0,Y 552.088,Z 455.711,A -85,B 0,C 180,E1 -3442.451,E2 -3442.451} C_VEL
LIN {X 0,Y 552.149,Z 455.703,A -85,B 0,C 180,E1 -3445.352,E2 -3445.352} C_VEL
LIN {X 0,Y 552.119,Z 455.703,A -85,B 0,C 180,E1 -3448.098,E2 -3448.098} C_VEL
LIN {X 0,Y 552.106,Z 455.705,A -85,B 0,C 180,E1 -3450.629,E2 -3450.629} C_VEL
LIN {X 0,Y 552.123,Z 455.708,A -85,B 0,C 180,E1 -3453.186,E2 -3453.186} C_VEL
LIN {X 0,Y 552.118,Z 455.704,A -85,B 0,C 180,E1 -3453.809,E2 -3453.809} C_VEL
LIN {X 0,Y 551.484,Z 455.787,A -85,B 0,C 180,E1 -3454.418,E2 -3454.418} C_VEL
LIN {X 0,Y 548.657,Z 456.146,A -85,B 0,C 180,E1 -3455.406,E2 -3455.406} C_VEL
LIN {X 0,Y 546.232,Z 456.452,A -85,B 0,C 180,E1 -3456.201,E2 -3456.201} C_VEL
LIN {X 0,Y 545.16,Z 456.581,A -85,B 0,C 180,E1 -3456.815,E2 -3456.815} C_VEL
LIN {X 0,Y 545.058,Z 456.59,A -85,B 0,C 180,E1 -3457.023,E2 -3457.023} C_VEL
LIN {X 0,Y 545.07,Z 456.575,A -85,B 0,C 180,E1 -3460.143,E2 -3460.143} C_VEL
LIN {X 0,Y 545.058,Z 456.588,A -85,B 0,C 180,E1 -3462.698,E2 -3462.698} C_VEL
LIN {X 0,Y 545.06,Z 456.589,A -85,B 0,C 180,E1 -3465.168,E2 -3465.168} C_VEL
LIN {X 0,Y 545.08,Z 456.578,A -85,B 0,C 180,E1 -3467.899,E2 -3467.899} C_VEL
LIN {X 0,Y 545.083,Z 456.589,A -85,B 0,C 180,E1 -3470.82,E2 -3470.82} C_VEL
LIN {X 0,Y 545.049,Z 456.579,A -85,B 0,C 180,E1 -3473.621,E2 -3473.621} C_VEL
LIN {X 0,Y 545.069,Z 456.573,A -85,B 0,C 180,E1 -3476.329,E2 -3476.329} C_VEL
LIN {X 0,Y 545.068,Z 456.59,A -85,B 0,C 180,E1 -3478.953,E2 -3478.953} C_VEL
LIN {X 0,Y 545.102,Z 456.578,A -85,B 0,C 180,E1 -3481.508,E2 -3481.508} C_VEL
LIN {X 0,Y 545.096,Z 456.579,A -85,B 0,C 180,E1 -3484.492,E2 -3484.492} C_VEL
LIN {X 0,Y 545.04,Z 456.589,A -85,B 0,C 180,E1 -3487.243,E2 -3487.243} C_VEL
LIN {X 0,Y 545.123,Z 456.579,A -85,B 0,C 180,E1 -3490.416,E2 -3490.416} C_VEL
LIN {X 0,Y 545.069,Z 456.572,A -85,B 0,C 180,E1 -3493.521,E2 -3493.521} C_VEL
LIN {X 0,Y 545.169,Z 456.748,A -85,B 0,C 180,E1 -3495.749,E2 -3495.749} C_VEL
LIN {X 0,Y 545.449,Z 457.97,A -85,B 0,C 180,E1 -3495.877,E2 -3495.877} C_VEL
LIN {X 0,Y 546.549,Z 461.934,A -85,B 0,C 180,E1 -3495.966,E2 -3495.966} C_VEL
LIN {X 0,Y 546.311,Z 536.302,A -85,B 0,C 180,E1 -3496.966,E2 -3496.966} C_VEL
LIN {X 0,Y 546.215,Z 549.457,A -85,B 0,C 180,E1 -3497.295,E2 -3497.295} C_VEL
LIN {X 0,Y 546.058,Z 561.166,A -85,B 0,C 180,E1 -3497.725,E2 -3497.725} C_VEL
LIN {X 0,Y 545.895,Z 572.942,A -85,B 0,C 180,E1 -3498.308,E2 -3498.308} C_VEL
LIN {X 0,Y 545.672,Z 584.409,A -85,B 0,C 180,E1 -3499.049,E2 -3499.049} C_VEL
LIN {X 0,Y 545.45,Z 594.765,A -85,B 0,C 180,E1 -3499.889,E2 -3499.889} C_VEL
LIN {X 0,Y 545.259,Z 603.213,A -85,B 0,C 180,E1 -3500.729,E2 -3500.729} C_VEL
LIN {X 0,Y 545.108,Z 610.976,A -85,B 0,C 180,E1 -3501.66,E2 -3501.66} C_VEL
LIN {X 0,Y 544.947,Z 618.668,A -85,B 0,C 180,E1 -3502.795,E2 -3502.795} C_VEL
LIN {X 0,Y 544.879,Z 625.49,A -85,B 0,C 180,E1 -3504.077,E2 -3504.077} C_VEL
LIN {X 0,Y 544.708,Z 630.122,A -85,B 0,C 180,E1 -3505.189,E2 -3505.189} C_VEL
LIN {X 0,Y 544.711,Z 633.648,A -85,B 0,C 180,E1 -3506.301,E2 -3506.301} C_VEL
LIN {X 0,Y 544.673,Z 635.477,A -85,B 0,C 180,E1 -3507.042,E2 -3507.042} C_VEL
LIN {X 0,Y 544.6,Z 636.863,A -85,B 0,C 180,E1 -3507.781,E2 -3507.781} C_VEL
LIN {X 0,Y 544.576,Z 638.445,A -85,B 0,C 180,E1 -3509.261,E2 -3509.261} C_VEL
LIN {X 0,Y 544.575,Z 638.679,A -85,B 0,C 180,E1 -3510,E2 -3510} C_VEL
LIN {X 0,Y 544.583,Z 637.935,A -85,B 0,C 180,E1 -3511.479,E2 -3511.479} C_VEL
LIN {X 0,Y 544.673,Z 635.664,A -85,B 0,C 180,E1 -3512.958,E2 -3512.958} C_VEL
LIN {X 0,Y 544.756,Z 632.858,A -85,B 0,C 180,E1 -3514.069,E2 -3514.069} C_VEL
LIN {X 0,Y 544.724,Z 629.073,A -85,B 0,C 180,E1 -3515.182,E2 -3515.182} C_VEL
LIN {X 0,Y 544.845,Z 623.874,A -85,B 0,C 180,E1 -3516.354,E2 -3516.354} C_VEL
LIN {X 0,Y 544.979,Z 616.781,A -85,B 0,C 180,E1 -3517.596,E2 -3517.596} C_VEL
LIN {X 0,Y 545.169,Z 608.768,A -85,B 0,C 180,E1 -3518.712,E2 -3518.712} C_VEL
LIN {X 0,Y 545.323,Z 600.558,A -85,B 0,C 180,E1 -3519.645,E2 -3519.645} C_VEL
LIN {X 0,Y 545.584,Z 590.393,A -85,B 0,C 180,E1 -3520.577,E2 -3520.577} C_VEL
LIN {X 0,Y 545.813,Z 579.106,A -85,B 0,C 180,E1 -3521.405,E2 -3521.405} C_VEL
LIN {X 0,Y 545.963,Z 567.478,A -85,B 0,C 180,E1 -3522.074,E2 -3522.074} C_VEL
LIN {X 0,Y 546.133,Z 555.553,A -85,B 0,C 180,E1 -3522.589,E2 -3522.589} C_VEL
LIN {X 0,Y 546.275,Z 542.566,A -85,B 0,C 180,E1 -3522.987,E2 -3522.987} C_VEL
LIN {X 0,Y 546.369,Z 530.183,A -85,B 0,C 180,E1 -3523.222,E2 -3523.222} C_VEL
LIN {X 0,Y 546.484,Z 461.085,A -85,B 0,C 180,E1 -3524.138,E2 -3524.138} C_VEL
LIN {X 0,Y 545.294,Z 457.405,A -85,B 0,C 180,E1 -3524.246,E2 -3524.246} C_VEL
LIN {X 0,Y 545.147,Z 456.617,A -85,B 0,C 180,E1 -3524.394,E2 -3524.394} C_VEL
LIN {X 0,Y 545.095,Z 456.566,A -85,B 0,C 180,E1 -3527.427,E2 -3527.427} C_VEL
LIN {X 0,Y 545.098,Z 456.583,A -85,B 0,C 180,E1 -3530.371,E2 -3530.371} C_VEL
LIN {X 0,Y 545.081,Z 456.584,A -85,B 0,C 180,E1 -3533.559,E2 -3533.559} C_VEL
LIN {X 0,Y 545.081,Z 456.58,A -85,B 0,C 180,E1 -3536,E2 -3536} C_VEL
LIN {X 0,Y 545.09,Z 456.581,A -85,B 0,C 180,E1 -3538.747,E2 -3538.747} C_VEL
LIN {X 0,Y 545.078,Z 456.582,A -85,B 0,C 180,E1 -3541.682,E2 -3541.682} C_VEL
LIN {X 0,Y 545.075,Z 456.586,A -85,B 0,C 180,E1 -3544.563,E2 -3544.563} C_VEL
LIN {X 0,Y 545.038,Z 456.592,A -85,B 0,C 180,E1 -3547.303,E2 -3547.303} C_VEL
LIN {X 0,Y 545.072,Z 456.583,A -85,B 0,C 180,E1 -3550.141,E2 -3550.141} C_VEL
LIN {X 0,Y 545.083,Z 456.585,A -85,B 0,C 180,E1 -3553.105,E2 -3553.105} C_VEL
LIN {X 0,Y 545.062,Z 456.585,A -85,B 0,C 180,E1 -3556.223,E2 -3556.223} C_VEL
LIN {X 0,Y 545.092,Z 456.584,A -85,B 0,C 180,E1 -3558.886,E2 -3558.886} C_VEL
LIN {X 0,Y 545.049,Z 456.585,A -85,B 0,C 180,E1 -3561.762,E2 -3561.762} C_VEL
LIN {X 0,Y 545.06,Z 456.586,A -85,B 0,C 180,E1 -3564.533,E2 -3564.533} C_VEL
LIN {X 0,Y 545.076,Z 456.586,A -85,B 0,C 180,E1 -3567.212,E2 -3567.212} C_VEL
LIN {X 0,Y 545.095,Z 456.573,A -85,B 0,C 180,E1 -3569.812,E2 -3569.812} C_VEL
LIN {X 0,Y 545.094,Z 456.581,A -85,B 0,C 180,E1 -3572.824,E2 -3572.824} C_VEL
LIN {X 0,Y 545.044,Z 456.589,A -85,B 0,C 180,E1 -3575.63,E2 -3575.63} C_VEL
LIN {X 0,Y 545.061,Z 456.585,A -85,B 0,C 180,E1 -3578.836,E2 -3578.836} C_VEL
LIN {X 0,Y 545.077,Z 456.591,A -85,B 0,C 180,E1 -3581.195,E2 -3581.195} C_VEL
LIN {X 0,Y 545.068,Z 456.587,A -85,B 0,C 180,E1 -3583.521,E2 -3583.521} C_VEL
LIN {X 0,Y 545.086,Z 456.584,A -85,B 0,C 180,E1 -3585.82,E2 -3585.82} C_VEL
LIN {X 0,Y 545.123,Z 456.578,A -85,B 0,C 180,E1 -3588.849,E2 -3588.849} C_VEL
LIN {X 0,Y 545.125,Z 456.578,A -85,B 0,C 180,E1 -3591.847,E2 -3591.847} C_VEL
LIN {X 0,Y 545.201,Z 456.568,A -85,B 0,C 180,E1 -3594.823,E2 -3594.823} C_VEL
LIN {X 0,Y 545.186,Z 456.57,A -85,B 0,C 180,E1 -3597.784,E2 -3597.784} C_VEL
LIN {X 0,Y 545.207,Z 456.566,A -85,B 0,C 180,E1 -3600.739,E2 -3600.739} C_VEL
LIN {X 0,Y 545.169,Z 456.572,A -85,B 0,C 180,E1 -3602.956,E2 -3602.956} C_VEL
LIN {X 0,Y 545.163,Z 456.574,A -85,B 0,C 180,E1 -3605.92,E2 -3605.92} C_VEL
LIN {X 0,Y 545.118,Z 456.578,A -85,B 0,C 180,E1 -3608.9,E2 -3608.9} C_VEL
LIN {X 0,Y 545.126,Z 456.579,A -85,B 0,C 180,E1 -3611.904,E2 -3611.904} C_VEL
LIN {X 0,Y 545.076,Z 456.584,A -85,B 0,C 180,E1 -3614.944,E2 -3614.944} C_VEL
LIN {X 0,Y 545.074,Z 456.579,A -85,B 0,C 180,E1 -3618.026,E2 -3618.026} C_VEL
LIN {X 0,Y 545.09,Z 456.578,A -85,B 0,C 180,E1 -3620.372,E2 -3620.372} C_VEL
LIN {X 0,Y 545.082,Z 456.591,A -85,B 0,C 180,E1 -3623.559,E2 -3623.559} C_VEL
LIN {X 0,Y 545.081,Z 456.581,A -85,B 0,C 180,E1 -3626.001,E2 -3626.001} C_VEL
LIN {X 0,Y 545.085,Z 456.58,A -85,B 0,C 180,E1 -3628.75,E2 -3628.75} C_VEL
LIN {X 0,Y 545.071,Z 456.591,A -85,B 0,C 180,E1 -3631.683,E2 -3631.683} C_VEL
LIN {X 0,Y 545.079,Z 456.582,A -85,B 0,C 180,E1 -3634.563,E2 -3634.563} C_VEL
LIN {X 0,Y 545.033,Z 456.591,A -85,B 0,C 180,E1 -3637.304,E2 -3637.304} C_VEL
LIN {X 0,Y 545.069,Z 456.587,A -85,B 0,C 180,E1 -3640.142,E2 -3640.142} C_VEL
LIN {X 0,Y 545.073,Z 456.58,A -85,B 0,C 180,E1 -3643.107,E2 -3643.107} C_VEL
LIN {X 0,Y 545.061,Z 456.589,A -85,B 0,C 180,E1 -3646.225,E2 -3646.225} C_VEL
LIN {X 0,Y 545.098,Z 456.578,A -85,B 0,C 180,E1 -3648.888,E2 -3648.888} C_VEL
LIN {X 0,Y 545.052,Z 456.594,A -85,B 0,C 180,E1 -3651.764,E2 -3651.764} C_VEL
LIN {X 0,Y 545.049,Z 456.588,A -85,B 0,C 180,E1 -3654.534,E2 -3654.534} C_VEL
LIN {X 0,Y 545.068,Z 456.584,A -85,B 0,C 180,E1 -3657.212,E2 -3657.212} C_VEL
LIN {X 0,Y 545.065,Z 456.579,A -85,B 0,C 180,E1 -3659.811,E2 -3659.811} C_VEL
LIN {X 0,Y 545.128,Z 456.808,A -85,B 0,C 180,E1 -3662.034,E2 -3662.034} C_VEL
LIN {X 0,Y 547.255,Z 466.673,A -85,B 0,C 180,E1 -3663.29,E2 -3663.29} C_VEL
LIN {X 0,Y 547.005,Z 488.646,A -85,B 0,C 180,E1 -3665.814,E2 -3665.814} C_VEL
LIN {X 0,Y 546.572,Z 514.252,A -85,B 0,C 180,E1 -3668.701,E2 -3668.701} C_VEL
LIN {X 0,Y 546.231,Z 540.529,A -85,B 0,C 180,E1 -3671.626,E2 -3671.626} C_VEL
LIN {X 0,Y 545.753,Z 567.445,A -85,B 0,C 180,E1 -3674.694,E2 -3674.694} C_VEL
LIN {X 0,Y 545.69,Z 574.18,A -85,B 0,C 180,E1 -3675.421,E2 -3675.421} C_VEL
LIN {X 0,Y 546.577,Z 581.61,A -85,B 0,C 180,E1 -3675.552,E2 -3675.552} C_VEL
LIN {X 0,Y 546.25,Z 683.962,A -85,B 0,C 180,E1 -3676.918,E2 -3676.918} C_VEL
LIN {X 0,Y 546.108,Z 696.465,A -85,B 0,C 180,E1 -3677.221,E2 -3677.221} C_VEL
LIN {X 0,Y 545.917,Z 709.377,A -85,B 0,C 180,E1 -3677.689,E2 -3677.689} C_VEL
LIN {X 0,Y 545.73,Z 721.673,A -85,B 0,C 180,E1 -3678.3,E2 -3678.3} C_VEL
LIN {X 0,Y 545.521,Z 733.2,A -85,B 0,C 180,E1 -3679.046,E2 -3679.046} C_VEL
LIN {X 0,Y 545.259,Z 743.607,A -85,B 0,C 180,E1 -3679.886,E2 -3679.886} C_VEL
LIN {X 0,Y 545.084,Z 752.115,A -85,B 0,C 180,E1 -3680.726,E2 -3680.726} C_VEL
LIN {X 0,Y 544.977,Z 759.962,A -85,B 0,C 180,E1 -3681.658,E2 -3681.658} C_VEL
LIN {X 0,Y 544.823,Z 767.623,A -85,B 0,C 180,E1 -3682.775,E2 -3682.775} C_VEL
LIN {X 0,Y 544.776,Z 774.68,A -85,B 0,C 180,E1 -3684.076,E2 -3684.076} C_VEL
LIN {X 0,Y 544.629,Z 779.373,A -85,B 0,C 180,E1 -3685.189,E2 -3685.189} C_VEL
LIN {X 0,Y 544.669,Z 782.958,A -85,B 0,C 180,E1 -3686.301,E2 -3686.301} C_VEL
LIN {X 0,Y 544.65,Z 784.808,A -85,B 0,C 180,E1 -3687.041,E2 -3687.041} C_VEL
LIN {X 0,Y 544.546,Z 787.184,A -85,B 0,C 180,E1 -3688.521,E2 -3688.521} C_VEL
LIN {X 0,Y 544.541,Z 788,A -85,B 0,C 180,E1 -3690,E2 -3690} C_VEL
LIN {X 0,Y 544.546,Z 787.185,A -85,B 0,C 180,E1 -3691.479,E2 -3691.479} C_VEL
LIN {X 0,Y 544.65,Z 784.81,A -85,B 0,C 180,E1 -3692.959,E2 -3692.959} C_VEL
LIN {X 0,Y 544.683,Z 781.896,A -85,B 0,C 180,E1 -3694.069,E2 -3694.069} C_VEL
LIN {X 0,Y 544.654,Z 777.949,A -85,B 0,C 180,E1 -3695.182,E2 -3695.182} C_VEL
LIN {X 0,Y 544.739,Z 772.704,A -85,B 0,C 180,E1 -3696.328,E2 -3696.328} C_VEL
LIN {X 0,Y 544.836,Z 766.468,A -85,B 0,C 180,E1 -3697.411,E2 -3697.411} C_VEL
LIN {X 0,Y 545.006,Z 758.479,A -85,B 0,C 180,E1 -3698.528,E2 -3698.528} C_VEL
LIN {X 0,Y 545.152,Z 750.336,A -85,B 0,C 180,E1 -3699.46,E2 -3699.46} C_VEL
LIN {X 0,Y 545.34,Z 740.401,A -85,B 0,C 180,E1 -3700.394,E2 -3700.394} C_VEL
LIN {X 0,Y 545.579,Z 729.543,A -85,B 0,C 180,E1 -3701.211,E2 -3701.211} C_VEL
LIN {X 0,Y 545.767,Z 718.178,A -85,B 0,C 180,E1 -3701.89,E2 -3701.89} C_VEL
LIN {X 0,Y 545.931,Z 705.982,A -85,B 0,C 180,E1 -3702.452,E2 -3702.452} C_VEL
LIN {X 0,Y 546.09,Z 693.186,A -85,B 0,C 180,E1 -3702.874,E2 -3702.874} C_VEL
LIN {X 0,Y 546.259,Z 679.621,A -85,B 0,C 180,E1 -3703.153,E2 -3703.153} C_VEL
LIN {X 0,Y 546.485,Z 580.332,A -85,B 0,C 180,E1 -3704.468,E2 -3704.468} C_VEL
LIN {X 0,Y 545.663,Z 573.926,A -85,B 0,C 180,E1 -3704.593,E2 -3704.593} C_VEL
LIN {X 0,Y 546.072,Z 547.157,A -85,B 0,C 180,E1 -3707.617,E2 -3707.617} C_VEL
LIN {X 0,Y 546.476,Z 523.025,A -85,B 0,C 180,E1 -3710.318,E2 -3710.318} C_VEL
LIN {X 0,Y 546.896,Z 496.668,A -85,B 0,C 180,E1 -3713.275,E2 -3713.275} C_VEL
LIN {X 0,Y 547.274,Z 470.217,A -85,B 0,C 180,E1 -3716.297,E2 -3716.297} C_VEL
LIN {X 0,Y 547.06,Z 465.188,A -85,B 0,C 180,E1 -3716.89,E2 -3716.89} C_VEL
LIN {X 0,Y 545.137,Z 456.717,A -85,B 0,C 180,E1 -3717.992,E2 -3717.992} C_VEL
LIN {X 0,Y 545.067,Z 456.583,A -85,B 0,C 180,E1 -3721.047,E2 -3721.047} C_VEL
LIN {X 0,Y 545.064,Z 456.586,A -85,B 0,C 180,E1 -3723.671,E2 -3723.671} C_VEL
LIN {X 0,Y 545.068,Z 456.583,A -85,B 0,C 180,E1 -3726.925,E2 -3726.925} C_VEL
LIN {X 0,Y 545.09,Z 456.585,A -85,B 0,C 180,E1 -3730.139,E2 -3730.139} C_VEL
LIN {X 0,Y 545.083,Z 456.583,A -85,B 0,C 180,E1 -3733.105,E2 -3733.105} C_VEL
LIN {X 0,Y 545.062,Z 456.585,A -85,B 0,C 180,E1 -3736.223,E2 -3736.223} C_VEL
LIN {X 0,Y 545.092,Z 456.582,A -85,B 0,C 180,E1 -3738.886,E2 -3738.886} C_VEL
LIN {X 0,Y 545.048,Z 456.587,A -85,B 0,C 180,E1 -3741.762,E2 -3741.762} C_VEL
LIN {X 0,Y 545.06,Z 456.59,A -85,B 0,C 180,E1 -3744.533,E2 -3744.533} C_VEL
LIN {X 0,Y 545.076,Z 456.58,A -85,B 0,C 180,E1 -3747.212,E2 -3747.212} C_VEL
LIN {X 0,Y 545.094,Z 456.582,A -85,B 0,C 180,E1 -3749.812,E2 -3749.812} C_VEL
LIN {X 0,Y 545.093,Z 456.578,A -85,B 0,C 180,E1 -3752.824,E2 -3752.824} C_VEL
LIN {X 0,Y 545.043,Z 456.586,A -85,B 0,C 180,E1 -3755.63,E2 -3755.63} C_VEL
LIN {X 0,Y 545.06,Z 456.585,A -85,B 0,C 180,E1 -3758.836,E2 -3758.836} C_VEL
LIN {X 0,Y 545.075,Z 456.576,A -85,B 0,C 180,E1 -3761.195,E2 -3761.195} C_VEL
LIN {X 0,Y 545.067,Z 456.582,A -85,B 0,C 180,E1 -3763.521,E2 -3763.521} C_VEL
LIN {X 0,Y 545.086,Z 456.582,A -85,B 0,C 180,E1 -3765.82,E2 -3765.82} C_VEL
LIN {X 0,Y 545.123,Z 456.578,A -85,B 0,C 180,E1 -3768.849,E2 -3768.849} C_VEL
LIN {X 0,Y 545.126,Z 456.577,A -85,B 0,C 180,E1 -3771.847,E2 -3771.847} C_VEL
LIN {X 0,Y 545.201,Z 456.568,A -85,B 0,C 180,E1 -3774.823,E2 -3774.823} C_VEL
LIN {X 0,Y 545.186,Z 456.568,A -85,B 0,C 180,E1 -3777.784,E2 -3777.784} C_VEL
LIN {X 0,Y 545.208,Z 456.571,A -85,B 0,C 180,E1 -3780.739,E2 -3780.739} C_VEL
LIN {X 0,Y 545.169,Z 456.573,A -85,B 0,C 180,E1 -3782.956,E2 -3782.956} C_VEL
LIN {X 0,Y 545.169,Z 456.571,A -85,B 0,C 180,E1 -3785.92,E2 -3785.92} C_VEL
LIN {X 0,Y 545.119,Z 456.579,A -85,B 0,C 180,E1 -3788.9,E2 -3788.9} C_VEL
LIN {X 0,Y 545.126,Z 456.576,A -85,B 0,C 180,E1 -3791.904,E2 -3791.904} C_VEL
LIN {X 0,Y 545.076,Z 456.585,A -85,B 0,C 180,E1 -3794.944,E2 -3794.944} C_VEL
LIN {X 0,Y 545.075,Z 456.582,A -85,B 0,C 180,E1 -3798.026,E2 -3798.026} C_VEL
LIN {X 0,Y 545.09,Z 456.584,A -85,B 0,C 180,E1 -3800.372,E2 -3800.372} C_VEL
LIN {X 0,Y 545.083,Z 456.581,A -85,B 0,C 180,E1 -3803.559,E2 -3803.559} C_VEL
LIN {X 0,Y 545.081,Z 456.582,A -85,B 0,C 180,E1 -3806.001,E2 -3806.001} C_VEL
LIN {X 0,Y 545.086,Z 456.585,A -85,B 0,C 180,E1 -3808.75,E2 -3808.75} C_VEL
LIN {X 0,Y 545.071,Z 456.576,A -85,B 0,C 180,E1 -3811.683,E2 -3811.683} C_VEL
LIN {X 0,Y 545.079,Z 456.585,A -85,B 0,C 180,E1 -3814.563,E2 -3814.563} C_VEL
LIN {X 0,Y 545.058,Z 456.59,A -85,B 0,C 180,E1 -3817.023,E2 -3817.023} C_VEL
LIN {X 0,Y 544.351,Z 456.674,A -85,B 0,C 180,E1 -3817.639,E2 -3817.639} C_VEL
LIN {X 0,Y 541.488,Z 457.033,A -85,B 0,C 180,E1 -3818.64,E2 -3818.64} C_VEL
LIN {X 0,Y 539.102,Z 457.322,A -85,B 0,C 180,E1 -3819.446,E2 -3819.446} C_VEL
LIN {X 0,Y 538.093,Z 457.444,A -85,B 0,C 180,E1 -3820.068,E2 -3820.068} C_VEL
LIN {X 0,Y 538.017,Z 457.454,A -85,B 0,C 180,E1 -3820.279,E2 -3820.279} C_VEL
LIN {X 0,Y 538.022,Z 457.47,A -85,B 0,C 180,E1 -3822.988,E2 -3822.988} C_VEL
LIN {X 0,Y 538.026,Z 457.458,A -85,B 0,C 180,E1 -3825.926,E2 -3825.926} C_VEL
LIN {X 0,Y 538.049,Z 457.464,A -85,B 0,C 180,E1 -3829.225,E2 -3829.225} C_VEL
LIN {X 0,Y 537.993,Z 457.464,A -85,B 0,C 180,E1 -3832.123,E2 -3832.123} C_VEL
LIN {X 0,Y 538.011,Z 457.455,A -85,B 0,C 180,E1 -3834.918,E2 -3834.918} C_VEL
LIN {X 0,Y 538.031,Z 457.461,A -85,B 0,C 180,E1 -3837.619,E2 -3837.619} C_VEL
LIN {X 0,Y 538.019,Z 457.463,A -85,B 0,C 180,E1 -3840.24,E2 -3840.24} C_VEL
LIN {X 0,Y 538.058,Z 457.455,A -85,B 0,C 180,E1 -3842.797,E2 -3842.797} C_VEL
LIN {X 0,Y 538.05,Z 457.466,A -85,B 0,C 180,E1 -3845.293,E2 -3845.293} C_VEL
LIN {X 0,Y 538.025,Z 457.459,A -85,B 0,C 180,E1 -3848.547,E2 -3848.547} C_VEL
LIN {X 0,Y 538.04,Z 457.461,A -85,B 0,C 180,E1 -3850.941,E2 -3850.941} C_VEL
LIN {X 0,Y 538.021,Z 457.445,A -85,B 0,C 180,E1 -3853.299,E2 -3853.299} C_VEL
LIN {X 0,Y 538.143,Z 457.579,A -85,B 0,C 180,E1 -3855.542,E2 -3855.542} C_VEL
LIN {X 0,Y 538.292,Z 458.388,A -85,B 0,C 180,E1 -3855.661,E2 -3855.661} C_VEL
LIN {X 0,Y 539.674,Z 462.543,A -85,B 0,C 180,E1 -3855.777,E2 -3855.777} C_VEL
LIN {X 0,Y 539.444,Z 537.321,A -85,B 0,C 180,E1 -3856.797,E2 -3856.797} C_VEL
LIN {X 0,Y 539.348,Z 550.466,A -85,B 0,C 180,E1 -3857.13,E2 -3857.13} C_VEL
LIN {X 0,Y 539.192,Z 562.168,A -85,B 0,C 180,E1 -3857.567,E2 -3857.567} C_VEL
LIN {X 0,Y 539.021,Z 573.94,A -85,B 0,C 180,E1 -3858.157,E2 -3858.157} C_VEL
LIN {X 0,Y 538.782,Z 585.403,A -85,B 0,C 180,E1 -3858.907,E2 -3858.907} C_VEL
LIN {X 0,Y 538.535,Z 595.759,A -85,B 0,C 180,E1 -3859.758,E2 -3859.758} C_VEL
LIN {X 0,Y 538.325,Z 604.205,A -85,B 0,C 180,E1 -3860.608,E2 -3860.608} C_VEL
LIN {X 0,Y 538.174,Z 611.964,A -85,B 0,C 180,E1 -3861.552,E2 -3861.552} C_VEL
LIN {X 0,Y 537.981,Z 619.66,A -85,B 0,C 180,E1 -3862.701,E2 -3862.701} C_VEL
LIN {X 0,Y 537.89,Z 626.479,A -85,B 0,C 180,E1 -3864,E2 -3864} C_VEL
LIN {X 0,Y 537.702,Z 631.111,A -85,B 0,C 180,E1 -3865.127,E2 -3865.127} C_VEL
LIN {X 0,Y 537.695,Z 634.638,A -85,B 0,C 180,E1 -3866.253,E2 -3866.253} C_VEL
LIN {X 0,Y 537.652,Z 636.466,A -85,B 0,C 180,E1 -3867.003,E2 -3867.003} C_VEL
LIN {X 0,Y 537.597,Z 637.849,A -85,B 0,C 180,E1 -3867.752,E2 -3867.752} C_VEL
LIN {X 0,Y 537.571,Z 639.43,A -85,B 0,C 180,E1 -3869.251,E2 -3869.251} C_VEL
LIN {X 0,Y 537.567,Z 639.664,A -85,B 0,C 180,E1 -3870,E2 -3870} C_VEL
LIN {X 0,Y 537.571,Z 639.486,A -85,B 0,C 180,E1 -3870.749,E2 -3870.749} C_VEL
LIN {X 0,Y 537.597,Z 637.977,A -85,B 0,C 180,E1 -3872.248,E2 -3872.248} C_VEL
LIN {X 0,Y 537.651,Z 636.65,A -85,B 0,C 180,E1 -3872.997,E2 -3872.997} C_VEL
LIN {X 0,Y 537.744,Z 633.846,A -85,B 0,C 180,E1 -3874.122,E2 -3874.122} C_VEL
LIN {X 0,Y 537.749,Z 630.057,A -85,B 0,C 180,E1 -3875.249,E2 -3875.249} C_VEL
LIN {X 0,Y 537.854,Z 624.888,A -85,B 0,C 180,E1 -3876.431,E2 -3876.431} C_VEL
LIN {X 0,Y 538.024,Z 617.762,A -85,B 0,C 180,E1 -3877.694,E2 -3877.694} C_VEL
LIN {X 0,Y 538.243,Z 609.749,A -85,B 0,C 180,E1 -3878.825,E2 -3878.825} C_VEL
LIN {X 0,Y 538.399,Z 601.541,A -85,B 0,C 180,E1 -3879.77,E2 -3879.77} C_VEL
LIN {X 0,Y 538.686,Z 591.371,A -85,B 0,C 180,E1 -3880.714,E2 -3880.714} C_VEL
LIN {X 0,Y 538.943,Z 581.054,A -85,B 0,C 180,E1 -3881.486,E2 -3881.486} C_VEL
LIN {X 0,Y 539.069,Z 570.422,A -85,B 0,C 180,E1 -3882.126,E2 -3882.126} C_VEL
LIN {X 0,Y 539.216,Z 559.034,A -85,B 0,C 180,E1 -3882.657,E2 -3882.657} C_VEL
LIN {X 0,Y 539.356,Z 546.267,A -85,B 0,C 180,E1 -3883.085,E2 -3883.085} C_VEL
LIN {X 0,Y 539.473,Z 534.165,A -85,B 0,C 180,E1 -3883.346,E2 -3883.346} C_VEL
LIN {X 0,Y 539.614,Z 462.43,A -85,B 0,C 180,E1 -3884.316,E2 -3884.316} C_VEL
LIN {X 0,Y 538.26,Z 458.27,A -85,B 0,C 180,E1 -3884.438,E2 -3884.438} C_VEL
LIN {X 0,Y 538.115,Z 457.487,A -85,B 0,C 180,E1 -3884.607,E2 -3884.607} C_VEL
LIN {X 0,Y 538.062,Z 457.44,A -85,B 0,C 180,E1 -3887.54,E2 -3887.54} C_VEL
LIN {X 0,Y 538.042,Z 457.466,A -85,B 0,C 180,E1 -3890.651,E2 -3890.651} C_VEL
LIN {X 0,Y 538.004,Z 457.464,A -85,B 0,C 180,E1 -3893.888,E2 -3893.888} C_VEL
LIN {X 0,Y 538.043,Z 457.458,A -85,B 0,C 180,E1 -3896.366,E2 -3896.366} C_VEL
LIN {X 0,Y 538.031,Z 457.463,A -85,B 0,C 180,E1 -3898.933,E2 -3898.933} C_VEL
LIN {X 0,Y 538.027,Z 457.459,A -85,B 0,C 180,E1 -3901.889,E2 -3901.889} C_VEL
LIN {X 0,Y 538.025,Z 457.465,A -85,B 0,C 180,E1 -3904.619,E2 -3904.619} C_VEL
LIN {X 0,Y 538.005,Z 457.468,A -85,B 0,C 180,E1 -3907.17,E2 -3907.17} C_VEL
LIN {X 0,Y 538.028,Z 457.462,A -85,B 0,C 180,E1 -3909.795,E2 -3909.795} C_VEL
LIN {X 0,Y 538.021,Z 457.462,A -85,B 0,C 180,E1 -3912.785,E2 -3912.785} C_VEL
LIN {X 0,Y 538.025,Z 457.462,A -85,B 0,C 180,E1 -3915.925,E2 -3915.925} C_VEL
LIN {X 0,Y 538.047,Z 457.457,A -85,B 0,C 180,E1 -3919.251,E2 -3919.251} C_VEL
LIN {X 0,Y 537.988,Z 457.463,A -85,B 0,C 180,E1 -3922.122,E2 -3922.122} C_VEL
LIN {X 0,Y 538.016,Z 457.468,A -85,B 0,C 180,E1 -3924.917,E2 -3924.917} C_VEL
LIN {X 0,Y 538.025,Z 457.457,A -85,B 0,C 180,E1 -3927.618,E2 -3927.618} C_VEL
LIN {X 0,Y 538.036,Z 457.45,A -85,B 0,C 180,E1 -3930.24,E2 -3930.24} C_VEL
LIN {X 0,Y 538.064,Z 457.456,A -85,B 0,C 180,E1 -3932.796,E2 -3932.796} C_VEL
LIN {X 0,Y 538.041,Z 457.467,A -85,B 0,C 180,E1 -3935.292,E2 -3935.292} C_VEL
LIN {X 0,Y 538.006,Z 457.461,A -85,B 0,C 180,E1 -3938.041,E2 -3938.041} C_VEL
LIN {X 0,Y 538.032,Z 457.464,A -85,B 0,C 180,E1 -3940.94,E2 -3940.94} C_VEL
LIN {X 0,Y 538.019,Z 457.467,A -85,B 0,C 180,E1 -3943.299,E2 -3943.299} C_VEL
LIN {X 0,Y 538.054,Z 457.462,A -85,B 0,C 180,E1 -3945.63,E2 -3945.63} C_VEL
LIN {X 0,Y 538.08,Z 457.454,A -85,B 0,C 180,E1 -3948.702,E2 -3948.702} C_VEL
LIN {X 0,Y 538.082,Z 457.456,A -85,B 0,C 180,E1 -3951.739,E2 -3951.739} C_VEL
LIN {X 0,Y 538.157,Z 457.445,A -85,B 0,C 180,E1 -3954.755,E2 -3954.755} C_VEL
LIN {X 0,Y 538.158,Z 457.446,A -85,B 0,C 180,E1 -3957.755,E2 -3957.755} C_VEL
LIN {X 0,Y 538.177,Z 457.442,A -85,B 0,C 180,E1 -3960.748,E2 -3960.748} C_VEL
LIN {X 0,Y 538.135,Z 457.448,A -85,B 0,C 180,E1 -3962.994,E2 -3962.994} C_VEL
LIN {X 0,Y 538.115,Z 457.451,A -85,B 0,C 180,E1 -3965.997,E2 -3965.997} C_VEL
LIN {X 0,Y 538.068,Z 457.458,A -85,B 0,C 180,E1 -3969.018,E2 -3969.018} C_VEL
LIN {X 0,Y 538.074,Z 457.456,A -85,B 0,C 180,E1 -3972.063,E2 -3972.063} C_VEL
LIN {X 0,Y 538.036,Z 457.463,A -85,B 0,C 180,E1 -3975.144,E2 -3975.144} C_VEL
LIN {X 0,Y 538.026,Z 457.454,A -85,B 0,C 180,E1 -3978.27,E2 -3978.27} C_VEL
LIN {X 0,Y 538.033,Z 457.457,A -85,B 0,C 180,E1 -3980.652,E2 -3980.652} C_VEL
LIN {X 0,Y 538.015,Z 457.467,A -85,B 0,C 180,E1 -3983.888,E2 -3983.888} C_VEL
LIN {X 0,Y 538.042,Z 457.454,A -85,B 0,C 180,E1 -3986.367,E2 -3986.367} C_VEL
LIN {X 0,Y 538.049,Z 457.457,A -85,B 0,C 180,E1 -3988.939,E2 -3988.939} C_VEL
LIN {X 0,Y 538.021,Z 457.465,A -85,B 0,C 180,E1 -3991.891,E2 -3991.891} C_VEL
LIN {X 0,Y 538.028,Z 457.46,A -85,B 0,C 180,E1 -3994.622,E2 -3994.622} C_VEL
LIN {X 0,Y 538.002,Z 457.466,A -85,B 0,C 180,E1 -3997.171,E2 -3997.171} C_VEL
LIN {X 0,Y 538.025,Z 457.471,A -85,B 0,C 180,E1 -3999.797,E2 -3999.797} C_VEL
LIN {X 0,Y 538.014,Z 457.458,A -85,B 0,C 180,E1 -4002.787,E2 -4002.787} C_VEL
LIN {X 0,Y 538.028,Z 457.457,A -85,B 0,C 180,E1 -4005.141,E2 -4005.141} C_VEL
LIN {X 0,Y 538.038,Z 457.46,A -85,B 0,C 180,E1 -4008.229,E2 -4008.229} C_VEL
LIN {X 0,Y 538.056,Z 457.459,A -85,B 0,C 180,E1 -4010.412,E2 -4010.412} C_VEL
LIN {X 0,Y 538.025,Z 457.461,A -85,B 0,C 180,E1 -4013.068,E2 -4013.068} C_VEL
LIN {X 0,Y 538.022,Z 457.469,A -85,B 0,C 180,E1 -4015.828,E2 -4015.828} C_VEL
LIN {X 0,Y 538.021,Z 457.462,A -85,B 0,C 180,E1 -4018.5,E2 -4018.5} C_VEL
LIN {X 0,Y 538.061,Z 457.502,A -85,B 0,C 180,E1 -4021.74,E2 -4021.74} C_VEL
LIN {X 0,Y 538.166,Z 458.044,A -85,B 0,C 180,E1 -4021.905,E2 -4021.905} C_VEL
LIN {X 0,Y 540.271,Z 467.547,A -85,B 0,C 180,E1 -4023.126,E2 -4023.126} C_VEL
LIN {X 0,Y 540.159,Z 483.441,A -85,B 0,C 180,E1 -4024.986,E2 -4024.986} C_VEL
LIN {X 0,Y 539.768,Z 506.086,A -85,B 0,C 180,E1 -4027.586,E2 -4027.586} C_VEL
LIN {X 0,Y 539.337,Z 530.876,A -85,B 0,C 180,E1 -4030.395,E2 -4030.395} C_VEL
LIN {X 0,Y 538.983,Z 555.393,A -85,B 0,C 180,E1 -4033.135,E2 -4033.135} C_VEL
LIN {X 0,Y 538.693,Z 573.921,A -85,B 0,C 180,E1 -4035.214,E2 -4035.214} C_VEL
LIN {X 0,Y 539.725,Z 582.263,A -85,B 0,C 180,E1 -4035.373,E2 -4035.373} C_VEL
LIN {X 0,Y 539.33,Z 683.961,A -85,B 0,C 180,E1 -4036.747,E2 -4036.747} C_VEL
LIN {X 0,Y 539.185,Z 697.227,A -85,B 0,C 180,E1 -4037.078,E2 -4037.078} C_VEL
LIN {X 0,Y 538.994,Z 709.376,A -85,B 0,C 180,E1 -4037.528,E2 -4037.528} C_VEL
LIN {X 0,Y 538.787,Z 720.794,A -85,B 0,C 180,E1 -4038.096,E2 -4038.096} C_VEL
LIN {X 0,Y 538.542,Z 731.906,A -85,B 0,C 180,E1 -4038.807,E2 -4038.807} C_VEL
LIN {X 0,Y 538.296,Z 742.539,A -85,B 0,C 180,E1 -4039.658,E2 -4039.658} C_VEL
LIN {X 0,Y 538.067,Z 752.115,A -85,B 0,C 180,E1 -4040.603,E2 -4040.603} C_VEL
LIN {X 0,Y 537.921,Z 759.962,A -85,B 0,C 180,E1 -4041.548,E2 -4041.548} C_VEL
LIN {X 0,Y 537.754,Z 767.623,A -85,B 0,C 180,E1 -4042.679,E2 -4042.679} C_VEL
LIN {X 0,Y 537.693,Z 774.68,A -85,B 0,C 180,E1 -4043.998,E2 -4043.998} C_VEL
LIN {X 0,Y 537.54,Z 779.373,A -85,B 0,C 180,E1 -4045.125,E2 -4045.125} C_VEL
LIN {X 0,Y 537.591,Z 782.958,A -85,B 0,C 180,E1 -4046.252,E2 -4046.252} C_VEL
LIN {X 0,Y 537.551,Z 784.807,A -85,B 0,C 180,E1 -4047.002,E2 -4047.002} C_VEL
LIN {X 0,Y 537.451,Z 787.183,A -85,B 0,C 180,E1 -4048.501,E2 -4048.501} C_VEL
LIN {X 0,Y 537.442,Z 788,A -85,B 0,C 180,E1 -4050,E2 -4050} C_VEL
LIN {X 0,Y 537.451,Z 787.184,A -85,B 0,C 180,E1 -4051.499,E2 -4051.499} C_VEL
LIN {X 0,Y 537.551,Z 784.81,A -85,B 0,C 180,E1 -4052.998,E2 -4052.998} C_VEL
LIN {X 0,Y 537.603,Z 781.896,A -85,B 0,C 180,E1 -4054.123,E2 -4054.123} C_VEL
LIN {X 0,Y 537.588,Z 777.949,A -85,B 0,C 180,E1 -4055.25,E2 -4055.25} C_VEL
LIN {X 0,Y 537.65,Z 773.081,A -85,B 0,C 180,E1 -4056.335,E2 -4056.335} C_VEL
LIN {X 0,Y 537.79,Z 766.468,A -85,B 0,C 180,E1 -4057.509,E2 -4057.509} C_VEL
LIN {X 0,Y 537.972,Z 758.479,A -85,B 0,C 180,E1 -4058.64,E2 -4058.64} C_VEL
LIN {X 0,Y 538.143,Z 750.336,A -85,B 0,C 180,E1 -4059.585,E2 -4059.585} C_VEL
LIN {X 0,Y 538.339,Z 740.401,A -85,B 0,C 180,E1 -4060.531,E2 -4060.531} C_VEL
LIN {X 0,Y 538.59,Z 730.595,A -85,B 0,C 180,E1 -4061.287,E2 -4061.287} C_VEL
LIN {X 0,Y 538.805,Z 719.701,A -85,B 0,C 180,E1 -4061.963,E2 -4061.963} C_VEL
LIN {X 0,Y 538.972,Z 707.109,A -85,B 0,C 180,E1 -4062.568,E2 -4062.568} C_VEL
LIN {X 0,Y 539.168,Z 694.098,A -85,B 0,C 180,E1 -4063.018,E2 -4063.018} C_VEL
LIN {X 0,Y 539.355,Z 681.124,A -85,B 0,C 180,E1 -4063.301,E2 -4063.301} C_VEL
LIN {X 0,Y 539.647,Z 581.357,A -85,B 0,C 180,E1 -4064.641,E2 -4064.641} C_VEL
LIN {X 0,Y 538.706,Z 573.928,A -85,B 0,C 180,E1 -4064.786,E2 -4064.786} C_VEL
LIN {X 0,Y 539.128,Z 545.207,A -85,B 0,C 180,E1 -4067.999,E2 -4067.999} C_VEL
LIN {X 0,Y 539.567,Z 518.618,A -85,B 0,C 180,E1 -4070.989,E2 -4070.989} C_VEL
LIN {X 0,Y 540.005,Z 492.693,A -85,B 0,C 180,E1 -4073.947,E2 -4073.947} C_VEL
LIN {X 0,Y 540.416,Z 469.332,A -85,B 0,C 180,E1 -4076.657,E2 -4076.657} C_VEL
LIN {X 0,Y 539.641,Z 464.544,A -85,B 0,C 180,E1 -4077.254,E2 -4077.254} C_VEL
LIN {X 0,Y 538.066,Z 457.593,A -85,B 0,C 180,E1 -4078.18,E2 -4078.18} C_VEL
LIN {X 0,Y 538.02,Z 457.46,A -85,B 0,C 180,E1 -4080.626,E2 -4080.626} C_VEL
LIN {X 0,Y 538.044,Z 457.458,A -85,B 0,C 180,E1 -4083.282,E2 -4083.282} C_VEL
LIN {X 0,Y 537.992,Z 457.471,A -85,B 0,C 180,E1 -4086.004,E2 -4086.004} C_VEL
LIN {X 0,Y 538.013,Z 457.463,A -85,B 0,C 180,E1 -4088.829,E2 -4088.829} C_VEL
LIN {X 0,Y 538.075,Z 457.454,A -85,B 0,C 180,E1 -4090.772,E2 -4090.772} C_VEL
LIN {X 0,Y 538.025,Z 457.469,A -85,B 0,C 180,E1 -4094.074,E2 -4094.074} C_VEL
LIN {X 0,Y 538.021,Z 457.458,A -85,B 0,C 180,E1 -4097.012,E2 -4097.012} C_VEL
LIN {X 0,Y 538.046,Z 457.458,A -85,B 0,C 180,E1 -4099.251,E2 -4099.251} C_VEL
LIN {X 0,Y 537.988,Z 457.47,A -85,B 0,C 180,E1 -4102.122,E2 -4102.122} C_VEL
LIN {X 0,Y 538.015,Z 457.463,A -85,B 0,C 180,E1 -4104.917,E2 -4104.917} C_VEL
LIN {X 0,Y 538.025,Z 457.459,A -85,B 0,C 180,E1 -4107.618,E2 -4107.618} C_VEL
LIN {X 0,Y 538.036,Z 457.468,A -85,B 0,C 180,E1 -4110.24,E2 -4110.24} C_VEL
LIN {X 0,Y 538.063,Z 457.454,A -85,B 0,C 180,E1 -4112.796,E2 -4112.796} C_VEL
LIN {X 0,Y 538.041,Z 457.458,A -85,B 0,C 180,E1 -4115.292,E2 -4115.292} C_VEL
LIN {X 0,Y 538.006,Z 457.467,A -85,B 0,C 180,E1 -4118.041,E2 -4118.041} C_VEL
LIN {X 0,Y 538.031,Z 457.455,A -85,B 0,C 180,E1 -4120.94,E2 -4120.94} C_VEL
LIN {X 0,Y 538.018,Z 457.46,A -85,B 0,C 180,E1 -4123.299,E2 -4123.299} C_VEL
LIN {X 0,Y 538.054,Z 457.457,A -85,B 0,C 180,E1 -4125.63,E2 -4125.63} C_VEL
LIN {X 0,Y 538.08,Z 457.458,A -85,B 0,C 180,E1 -4128.702,E2 -4128.702} C_VEL
LIN {X 0,Y 538.082,Z 457.454,A -85,B 0,C 180,E1 -4131.74,E2 -4131.74} C_VEL
LIN {X 0,Y 538.176,Z 457.444,A -85,B 0,C 180,E1 -4134.755,E2 -4134.755} C_VEL
LIN {X 0,Y 538.158,Z 457.443,A -85,B 0,C 180,E1 -4137.755,E2 -4137.755} C_VEL
LIN {X 0,Y 538.178,Z 457.447,A -85,B 0,C 180,E1 -4140.748,E2 -4140.748} C_VEL
LIN {X 0,Y 538.135,Z 457.448,A -85,B 0,C 180,E1 -4142.995,E2 -4142.995} C_VEL
LIN {X 0,Y 538.123,Z 457.449,A -85,B 0,C 180,E1 -4145.997,E2 -4145.997} C_VEL
LIN {X 0,Y 538.068,Z 457.455,A -85,B 0,C 180,E1 -4149.018,E2 -4149.018} C_VEL
LIN {X 0,Y 538.074,Z 457.455,A -85,B 0,C 180,E1 -4152.063,E2 -4152.063} C_VEL
LIN {X 0,Y 538.036,Z 457.459,A -85,B 0,C 180,E1 -4155.144,E2 -4155.144} C_VEL
LIN {X 0,Y 538.027,Z 457.462,A -85,B 0,C 180,E1 -4158.27,E2 -4158.27} C_VEL
LIN {X 0,Y 538.034,Z 457.468,A -85,B 0,C 180,E1 -4160.652,E2 -4160.652} C_VEL
LIN {X 0,Y 538.016,Z 457.461,A -85,B 0,C 180,E1 -4163.888,E2 -4163.888} C_VEL
LIN {X 0,Y 538.043,Z 457.462,A -85,B 0,C 180,E1 -4166.367,E2 -4166.367} C_VEL
LIN {X 0,Y 538.049,Z 457.457,A -85,B 0,C 180,E1 -4168.939,E2 -4168.939} C_VEL
LIN {X 0,Y 538.021,Z 457.453,A -85,B 0,C 180,E1 -4171.891,E2 -4171.891} C_VEL
LIN {X 0,Y 538.029,Z 457.464,A -85,B 0,C 180,E1 -4174.622,E2 -4174.622} C_VEL
LIN {X 0,Y 538.002,Z 457.467,A -85,B 0,C 180,E1 -4177.171,E2 -4177.171} C_VEL
LIN {X 0,Y 538.017,Z 457.454,A -85,B 0,C 180,E1 -4180.279,E2 -4180.279} C_VEL
LIN {X 0,Y 537.368,Z 457.544,A -85,B 0,C 180,E1 -4180.904,E2 -4180.904} C_VEL
LIN {X 0,Y 534.516,Z 457.902,A -85,B 0,C 180,E1 -4181.919,E2 -4181.919} C_VEL
LIN {X 0,Y 532.092,Z 458.205,A -85,B 0,C 180,E1 -4182.736,E2 -4182.736} C_VEL
LIN {X 0,Y 531.045,Z 458.335,A -85,B 0,C 180,E1 -4183.367,E2 -4183.367} C_VEL
LIN {X 0,Y 530.957,Z 458.343,A -85,B 0,C 180,E1 -4183.581,E2 -4183.581} C_VEL
LIN {X 0,Y 530.964,Z 458.341,A -85,B 0,C 180,E1 -4186.507,E2 -4186.507} C_VEL
LIN {X 0,Y 530.987,Z 458.343,A -85,B 0,C 180,E1 -4188.976,E2 -4188.976} C_VEL
LIN {X 0,Y 530.958,Z 458.342,A -85,B 0,C 180,E1 -4191.531,E2 -4191.531} C_VEL
LIN {X 0,Y 530.975,Z 458.33,A -85,B 0,C 180,E1 -4194.383,E2 -4194.383} C_VEL
LIN {X 0,Y 530.972,Z 458.338,A -85,B 0,C 180,E1 -4197.135,E2 -4197.135} C_VEL
LIN {X 0,Y 530.97,Z 458.342,A -85,B 0,C 180,E1 -4199.804,E2 -4199.804} C_VEL
LIN {X 0,Y 531.013,Z 458.33,A -85,B 0,C 180,E1 -4202.468,E2 -4202.468} C_VEL
LIN {X 0,Y 531.007,Z 458.34,A -85,B 0,C 180,E1 -4204.943,E2 -4204.943} C_VEL
LIN {X 0,Y 530.973,Z 458.336,A -85,B 0,C 180,E1 -4208.247,E2 -4208.247} C_VEL
LIN {X 0,Y 530.999,Z 458.341,A -85,B 0,C 180,E1 -4210.678,E2 -4210.678} C_VEL
LIN {X 0,Y 530.984,Z 458.318,A -85,B 0,C 180,E1 -4213.071,E2 -4213.071} C_VEL
LIN {X 0,Y 531.071,Z 458.455,A -85,B 0,C 180,E1 -4215.338,E2 -4215.338} C_VEL
LIN {X 0,Y 531.272,Z 459.314,A -85,B 0,C 180,E1 -4215.468,E2 -4215.468} C_VEL
LIN {X 0,Y 532.78,Z 463.814,A -85,B 0,C 180,E1 -4215.592,E2 -4215.592} C_VEL
LIN {X 0,Y 532.581,Z 538.341,A -85,B 0,C 180,E1 -4216.624,E2 -4216.624} C_VEL
LIN {X 0,Y 532.486,Z 551.475,A -85,B 0,C 180,E1 -4216.961,E2 -4216.961} C_VEL
LIN {X 0,Y 532.327,Z 563.17,A -85,B 0,C 180,E1 -4217.404,E2 -4217.404} C_VEL
LIN {X 0,Y 532.161,Z 575.265,A -85,B 0,C 180,E1 -4218.021,E2 -4218.021} C_VEL
LIN {X 0,Y 531.885,Z 586.399,A -85,B 0,C 180,E1 -4218.762,E2 -4218.762} C_VEL
LIN {X 0,Y 531.627,Z 596.752,A -85,B 0,C 180,E1 -4219.624,E2 -4219.624} C_VEL
LIN {X 0,Y 531.394,Z 605.199,A -85,B 0,C 180,E1 -4220.484,E2 -4220.484} C_VEL
LIN {X 0,Y 531.238,Z 612.955,A -85,B 0,C 180,E1 -4221.441,E2 -4221.441} C_VEL
LIN {X 0,Y 531.015,Z 620.651,A -85,B 0,C 180,E1 -4222.605,E2 -4222.605} C_VEL
LIN {X 0,Y 530.905,Z 627.469,A -85,B 0,C 180,E1 -4223.921,E2 -4223.921} C_VEL
LIN {X 0,Y 530.698,Z 632.101,A -85,B 0,C 180,E1 -4225.062,E2 -4225.062} C_VEL
LIN {X 0,Y 530.68,Z 635.628,A -85,B 0,C 180,E1 -4226.203,E2 -4226.203} C_VEL
LIN {X 0,Y 530.631,Z 637.455,A -85,B 0,C 180,E1 -4226.963,E2 -4226.963} C_VEL
LIN {X 0,Y 530.592,Z 638.835,A -85,B 0,C 180,E1 -4227.723,E2 -4227.723} C_VEL
LIN {X 0,Y 530.564,Z 640.416,A -85,B 0,C 180,E1 -4229.241,E2 -4229.241} C_VEL
LIN {X 0,Y 530.557,Z 640.65,A -85,B 0,C 180,E1 -4230,E2 -4230} C_VEL
LIN {X 0,Y 530.564,Z 640.471,A -85,B 0,C 180,E1 -4230.759,E2 -4230.759} C_VEL
LIN {X 0,Y 530.592,Z 638.961,A -85,B 0,C 180,E1 -4232.277,E2 -4232.277} C_VEL
LIN {X 0,Y 530.629,Z 637.637,A -85,B 0,C 180,E1 -4233.037,E2 -4233.037} C_VEL
LIN {X 0,Y 530.732,Z 634.833,A -85,B 0,C 180,E1 -4234.177,E2 -4234.177} C_VEL
LIN {X 0,Y 530.773,Z 631.039,A -85,B 0,C 180,E1 -4235.318,E2 -4235.318} C_VEL
LIN {X 0,Y 530.866,Z 625.895,A -85,B 0,C 180,E1 -4236.512,E2 -4236.512} C_VEL
LIN {X 0,Y 531.067,Z 618.745,A -85,B 0,C 180,E1 -4237.796,E2 -4237.796} C_VEL
LIN {X 0,Y 531.309,Z 610.731,A -85,B 0,C 180,E1 -4238.941,E2 -4238.941} C_VEL
LIN {X 0,Y 531.478,Z 602.523,A -85,B 0,C 180,E1 -4239.898,E2 -4239.898} C_VEL
LIN {X 0,Y 531.789,Z 592.351,A -85,B 0,C 180,E1 -4240.855,E2 -4240.855} C_VEL
LIN {X 0,Y 532.065,Z 582.033,A -85,B 0,C 180,E1 -4241.636,E2 -4241.636} C_VEL
LIN {X 0,Y 532.215,Z 570.137,A -85,B 0,C 180,E1 -4242.354,E2 -4242.354} C_VEL
LIN {X 0,Y 532.393,Z 557.628,A -85,B 0,C 180,E1 -4242.915,E2 -4242.915} C_VEL
LIN {X 0,Y 532.549,Z 544.502,A -85,B 0,C 180,E1 -4243.328,E2 -4243.328} C_VEL
LIN {X 0,Y 532.644,Z 532.078,A -85,B 0,C 180,E1 -4243.569,E2 -4243.569} C_VEL
LIN {X 0,Y 532.77,Z 463.814,A -85,B 0,C 180,E1 -4244.498,E2 -4244.498} C_VEL
LIN {X 0,Y 531.199,Z 459.11,A -85,B 0,C 180,E1 -4244.639,E2 -4244.639} C_VEL
LIN {X 0,Y 531.049,Z 458.383,A -85,B 0,C 180,E1 -4244.789,E2 -4244.789} C_VEL
LIN {X 0,Y 531.019,Z 458.317,A -85,B 0,C 180,E1 -4247.722,E2 -4247.722} C_VEL
LIN {X 0,Y 531.002,Z 458.342,A -85,B 0,C 180,E1 -4250.937,E2 -4250.937} C_VEL
LIN {X 0,Y 530.972,Z 458.341,A -85,B 0,C 180,E1 -4254.224,E2 -4254.224} C_VEL
LIN {X 0,Y 531.002,Z 458.335,A -85,B 0,C 180,E1 -4256.743,E2 -4256.743} C_VEL
LIN {X 0,Y 530.982,Z 458.344,A -85,B 0,C 180,E1 -4259.322,E2 -4259.322} C_VEL
LIN {X 0,Y 530.979,Z 458.337,A -85,B 0,C 180,E1 -4262.102,E2 -4262.102} C_VEL
LIN {X 0,Y 530.981,Z 458.346,A -85,B 0,C 180,E1 -4264.852,E2 -4264.852} C_VEL
LIN {X 0,Y 530.965,Z 458.342,A -85,B 0,C 180,E1 -4267.507,E2 -4267.507} C_VEL
LIN {X 0,Y 530.982,Z 458.34,A -85,B 0,C 180,E1 -4270.432,E2 -4270.432} C_VEL
LIN {X 0,Y 530.967,Z 458.344,A -85,B 0,C 180,E1 -4273.281,E2 -4273.281} C_VEL
LIN {X 0,Y 530.984,Z 458.341,A -85,B 0,C 180,E1 -4275.62,E2 -4275.62} C_VEL
LIN {X 0,Y 530.995,Z 458.336,A -85,B 0,C 180,E1 -4278.564,E2 -4278.564} C_VEL
LIN {X 0,Y 530.954,Z 458.343,A -85,B 0,C 180,E1 -4281.529,E2 -4281.529} C_VEL
LIN {X 0,Y 530.977,Z 458.339,A -85,B 0,C 180,E1 -4284.381,E2 -4284.381} C_VEL
LIN {X 0,Y 530.968,Z 458.343,A -85,B 0,C 180,E1 -4287.133,E2 -4287.133} C_VEL
LIN {X 0,Y 530.979,Z 458.33,A -85,B 0,C 180,E1 -4289.803,E2 -4289.803} C_VEL
LIN {X 0,Y 531.01,Z 458.332,A -85,B 0,C 180,E1 -4292.466,E2 -4292.466} C_VEL
LIN {X 0,Y 531,Z 458.341,A -85,B 0,C 180,E1 -4294.942,E2 -4294.942} C_VEL
LIN {X 0,Y 530.963,Z 458.338,A -85,B 0,C 180,E1 -4298.246,E2 -4298.246} C_VEL
LIN {X 0,Y 530.989,Z 458.339,A -85,B 0,C 180,E1 -4300.677,E2 -4300.677} C_VEL
LIN {X 0,Y 530.984,Z 458.342,A -85,B 0,C 180,E1 -4303.071,E2 -4303.071} C_VEL
LIN {X 0,Y 531.031,Z 458.34,A -85,B 0,C 180,E1 -4305.436,E2 -4305.436} C_VEL
LIN {X 0,Y 531.037,Z 458.331,A -85,B 0,C 180,E1 -4308.55,E2 -4308.55} C_VEL
LIN {X 0,Y 531.051,Z 458.334,A -85,B 0,C 180,E1 -4311.629,E2 -4311.629} C_VEL
LIN {X 0,Y 531.116,Z 458.322,A -85,B 0,C 180,E1 -4314.685,E2 -4314.685} C_VEL
LIN {X 0,Y 531.13,Z 458.321,A -85,B 0,C 180,E1 -4317.725,E2 -4317.725} C_VEL
LIN {X 0,Y 531.147,Z 458.318,A -85,B 0,C 180,E1 -4320.758,E2 -4320.758} C_VEL
LIN {X 0,Y 531.101,Z 458.325,A -85,B 0,C 180,E1 -4323.034,E2 -4323.034} C_VEL
LIN {X 0,Y 531.075,Z 458.327,A -85,B 0,C 180,E1 -4326.077,E2 -4326.077} C_VEL
LIN {X 0,Y 531.027,Z 458.336,A -85,B 0,C 180,E1 -4329.138,E2 -4329.138} C_VEL
LIN {X 0,Y 531.031,Z 458.332,A -85,B 0,C 180,E1 -4332.225,E2 -4332.225} C_VEL
LIN {X 0,Y 530.986,Z 458.344,A -85,B 0,C 180,E1 -4335.35,E2 -4335.35} C_VEL
LIN {X 0,Y 531.007,Z 458.334,A -85,B 0,C 180,E1 -4337.723,E2 -4337.723} C_VEL
LIN {X 0,Y 530.993,Z 458.335,A -85,B 0,C 180,E1 -4340.938,E2 -4340.938} C_VEL
LIN {X 0,Y 530.971,Z 458.34,A -85,B 0,C 180,E1 -4344.225,E2 -4344.225} C_VEL
LIN {X 0,Y 531.004,Z 458.329,A -85,B 0,C 180,E1 -4346.744,E2 -4346.744} C_VEL
LIN {X 0,Y 530.993,Z 458.34,A -85,B 0,C 180,E1 -4349.322,E2 -4349.322} C_VEL
LIN {X 0,Y 530.973,Z 458.339,A -85,B 0,C 180,E1 -4352.104,E2 -4352.104} C_VEL
LIN {X 0,Y 530.985,Z 458.337,A -85,B 0,C 180,E1 -4354.855,E2 -4354.855} C_VEL
LIN {X 0,Y 530.96,Z 458.347,A -85,B 0,C 180,E1 -4357.508,E2 -4357.508} C_VEL
LIN {X 0,Y 530.98,Z 458.34,A -85,B 0,C 180,E1 -4360.433,E2 -4360.433} C_VEL
LIN {X 0,Y 530.96,Z 458.342,A -85,B 0,C 180,E1 -4363.495,E2 -4363.495} C_VEL
LIN {X 0,Y 530.962,Z 458.343,A -85,B 0,C 180,E1 -4366.506,E2 -4366.506} C_VEL
LIN {X 0,Y 531.023,Z 458.335,A -85,B 0,C 180,E1 -4369.572,E2 -4369.572} C_VEL
LIN {X 0,Y 530.966,Z 458.34,A -85,B 0,C 180,E1 -4372.578,E2 -4372.578} C_VEL
LIN {X 0,Y 530.993,Z 458.341,A -85,B 0,C 180,E1 -4375.311,E2 -4375.311} C_VEL
LIN {X 0,Y 530.977,Z 458.345,A -85,B 0,C 180,E1 -4378.033,E2 -4378.033} C_VEL
LIN {X 0,Y 530.988,Z 458.332,A -85,B 0,C 180,E1 -4380.875,E2 -4380.875} C_VEL
LIN {X 0,Y 531.044,Z 458.56,A -85,B 0,C 180,E1 -4381.657,E2 -4381.657} C_VEL
LIN {X 0,Y 533.477,Z 470.204,A -85,B 0,C 180,E1 -4383.179,E2 -4383.179} C_VEL
LIN {X 0,Y 533.093,Z 491.733,A -85,B 0,C 180,E1 -4385.716,E2 -4385.716} C_VEL
LIN {X 0,Y 532.606,Z 517.705,A -85,B 0,C 180,E1 -4388.724,E2 -4388.724} C_VEL
LIN {X 0,Y 532.09,Z 546.351,A -85,B 0,C 180,E1 -4391.989,E2 -4391.989} C_VEL
LIN {X 0,Y 531.693,Z 573.459,A -85,B 0,C 180,E1 -4395.023,E2 -4395.023} C_VEL
LIN {X 0,Y 532.845,Z 582.735,A -85,B 0,C 180,E1 -4395.194,E2 -4395.194} C_VEL
LIN {X 0,Y 532.432,Z 683.827,A -85,B 0,C 180,E1 -4396.572,E2 -4396.572} C_VEL
LIN {X 0,Y 532.255,Z 696.419,A -85,B 0,C 180,E1 -4396.883,E2 -4396.883} C_VEL
LIN {X 0,Y 532.046,Z 709.375,A -85,B 0,C 180,E1 -4397.363,E2 -4397.363} C_VEL
LIN {X 0,Y 531.808,Z 721.311,A -85,B 0,C 180,E1 -4397.968,E2 -4397.968} C_VEL
LIN {X 0,Y 531.558,Z 733.196,A -85,B 0,C 180,E1 -4398.755,E2 -4398.755} C_VEL
LIN {X 0,Y 531.267,Z 743.607,A -85,B 0,C 180,E1 -4399.616,E2 -4399.616} C_VEL
LIN {X 0,Y 531.06,Z 752.115,A -85,B 0,C 180,E1 -4400.478,E2 -4400.478} C_VEL
LIN {X 0,Y 530.886,Z 759.962,A -85,B 0,C 180,E1 -4401.435,E2 -4401.435} C_VEL
LIN {X 0,Y 530.684,Z 767.622,A -85,B 0,C 180,E1 -4402.581,E2 -4402.581} C_VEL
LIN {X 0,Y 530.604,Z 774.68,A -85,B 0,C 180,E1 -4403.918,E2 -4403.918} C_VEL
LIN {X 0,Y 530.459,Z 779.373,A -85,B 0,C 180,E1 -4405.06,E2 -4405.06} C_VEL
LIN {X 0,Y 530.516,Z 782.958,A -85,B 0,C 180,E1 -4406.202,E2 -4406.202} C_VEL
LIN {X 0,Y 530.457,Z 784.807,A -85,B 0,C 180,E1 -4406.962,E2 -4406.962} C_VEL
LIN {X 0,Y 530.41,Z 786.194,A -85,B 0,C 180,E1 -4407.722,E2 -4407.722} C_VEL
LIN {X 0,Y 530.344,Z 787.786,A -85,B 0,C 180,E1 -4409.241,E2 -4409.241} C_VEL
LIN {X 0,Y 530.342,Z 788,A -85,B 0,C 180,E1 -4410,E2 -4410} C_VEL
LIN {X 0,Y 530.361,Z 787.184,A -85,B 0,C 180,E1 -4411.519,E2 -4411.519} C_VEL
LIN {X 0,Y 530.41,Z 786.196,A -85,B 0,C 180,E1 -4412.278,E2 -4412.278} C_VEL
LIN {X 0,Y 530.457,Z 784.81,A -85,B 0,C 180,E1 -4413.038,E2 -4413.038} C_VEL
LIN {X 0,Y 530.522,Z 781.896,A -85,B 0,C 180,E1 -4414.178,E2 -4414.178} C_VEL
LIN {X 0,Y 530.525,Z 777.948,A -85,B 0,C 180,E1 -4415.321,E2 -4415.321} C_VEL
LIN {X 0,Y 530.599,Z 772.263,A -85,B 0,C 180,E1 -4416.582,E2 -4416.582} C_VEL
LIN {X 0,Y 530.758,Z 765.236,A -85,B 0,C 180,E1 -4417.8,E2 -4417.8} C_VEL
LIN {X 0,Y 530.93,Z 756.994,A -85,B 0,C 180,E1 -4418.948,E2 -4418.948} C_VEL
LIN {X 0,Y 531.139,Z 748.542,A -85,B 0,C 180,E1 -4419.905,E2 -4419.905} C_VEL
LIN {X 0,Y 531.413,Z 738.094,A -85,B 0,C 180,E1 -4420.863,E2 -4420.863} C_VEL
LIN {X 0,Y 531.703,Z 727.138,A -85,B 0,C 180,E1 -4421.67,E2 -4421.67} C_VEL
LIN {X 0,Y 531.932,Z 716.409,A -85,B 0,C 180,E1 -4422.301,E2 -4422.301} C_VEL
LIN {X 0,Y 532.109,Z 704.765,A -85,B 0,C 180,E1 -4422.83,E2 -4422.83} C_VEL
LIN {X 0,Y 532.297,Z 692.186,A -85,B 0,C 180,E1 -4423.237,E2 -4423.237} C_VEL
LIN {X 0,Y 532.445,Z 679.454,A -85,B 0,C 180,E1 -4423.501,E2 -4423.501} C_VEL
LIN {X 0,Y 532.715,Z 581.534,A -85,B 0,C 180,E1 -4424.826,E2 -4424.826} C_VEL
LIN {X 0,Y 531.716,Z 573.449,A -85,B 0,C 180,E1 -4424.977,E2 -4424.977} C_VEL
LIN {X 0,Y 532.114,Z 544.77,A -85,B 0,C 180,E1 -4428.185,E2 -4428.185} C_VEL
LIN {X 0,Y 532.59,Z 517.701,A -85,B 0,C 180,E1 -4431.277,E2 -4431.277} C_VEL
LIN {X 0,Y 533.054,Z 493.115,A -85,B 0,C 180,E1 -4434.124,E2 -4434.124} C_VEL
LIN {X 0,Y 533.487,Z 470.197,A -85,B 0,C 180,E1 -4436.82,E2 -4436.82} C_VEL
LIN {X 0,Y 531.046,Z 458.52,A -85,B 0,C 180,E1 -4438.352,E2 -4438.352} C_VEL
LIN {X 0,Y 530.957,Z 458.341,A -85,B 0,C 180,E1 -4441.078,E2 -4441.078} C_VEL
LIN {X 0,Y 530.985,Z 458.34,A -85,B 0,C 180,E1 -4443.772,E2 -4443.772} C_VEL
LIN {X 0,Y 530.952,Z 458.345,A -85,B 0,C 180,E1 -4446.558,E2 -4446.558} C_VEL
LIN {X 0,Y 531.003,Z 458.34,A -85,B 0,C 180,E1 -4449.857,E2 -4449.857} C_VEL
LIN {X 0,Y 530.979,Z 458.346,A -85,B 0,C 180,E1 -4452.455,E2 -4452.455} C_VEL
LIN {X 0,Y 530.983,Z 458.334,A -85,B 0,C 180,E1 -4455.62,E2 -4455.62} C_VEL
LIN {X 0,Y 530.995,Z 458.342,A -85,B 0,C 180,E1 -4458.564,E2 -4458.564} C_VEL
LIN {X 0,Y 530.953,Z 458.34,A -85,B 0,C 180,E1 -4461.529,E2 -4461.529} C_VEL
LIN {X 0,Y 530.976,Z 458.347,A -85,B 0,C 180,E1 -4464.382,E2 -4464.382} C_VEL
LIN {X 0,Y 530.968,Z 458.337,A -85,B 0,C 180,E1 -4467.133,E2 -4467.133} C_VEL
LIN {X 0,Y 530.979,Z 458.341,A -85,B 0,C 180,E1 -4469.804,E2 -4469.804} C_VEL
LIN {X 0,Y 531.01,Z 458.336,A -85,B 0,C 180,E1 -4472.466,E2 -4472.466} C_VEL
LIN {X 0,Y 531,Z 458.337,A -85,B 0,C 180,E1 -4474.942,E2 -4474.942} C_VEL
LIN {X 0,Y 530.963,Z 458.347,A -85,B 0,C 180,E1 -4478.246,E2 -4478.246} C_VEL
LIN {X 0,Y 530.988,Z 458.335,A -85,B 0,C 180,E1 -4480.677,E2 -4480.677} C_VEL
LIN {X 0,Y 530.983,Z 458.337,A -85,B 0,C 180,E1 -4483.071,E2 -4483.071} C_VEL
LIN {X 0,Y 531.009,Z 458.335,A -85,B 0,C 180,E1 -4485.436,E2 -4485.436} C_VEL
LIN {X 0,Y 531.037,Z 458.336,A -85,B 0,C 180,E1 -4488.55,E2 -4488.55} C_VEL
LIN {X 0,Y 531.051,Z 458.329,A -85,B 0,C 180,E1 -4491.629,E2 -4491.629} C_VEL
LIN {X 0,Y 531.132,Z 458.322,A -85,B 0,C 180,E1 -4494.685,E2 -4494.685} C_VEL
LIN {X 0,Y 531.13,Z 458.319,A -85,B 0,C 180,E1 -4497.725,E2 -4497.725} C_VEL
LIN {X 0,Y 531.147,Z 458.322,A -85,B 0,C 180,E1 -4500.758,E2 -4500.758} C_VEL
LIN {X 0,Y 531.101,Z 458.324,A -85,B 0,C 180,E1 -4503.034,E2 -4503.034} C_VEL
LIN {X 0,Y 531.081,Z 458.327,A -85,B 0,C 180,E1 -4506.077,E2 -4506.077} C_VEL
LIN {X 0,Y 531.027,Z 458.331,A -85,B 0,C 180,E1 -4509.138,E2 -4509.138} C_VEL
LIN {X 0,Y 531.032,Z 458.334,A -85,B 0,C 180,E1 -4512.225,E2 -4512.225} C_VEL
LIN {X 0,Y 530.987,Z 458.335,A -85,B 0,C 180,E1 -4515.35,E2 -4515.35} C_VEL
LIN {X 0,Y 531.007,Z 458.334,A -85,B 0,C 180,E1 -4517.723,E2 -4517.723} C_VEL
LIN {X 0,Y 530.994,Z 458.341,A -85,B 0,C 180,E1 -4520.938,E2 -4520.938} C_VEL
LIN {X 0,Y 530.972,Z 458.34,A -85,B 0,C 180,E1 -4524.225,E2 -4524.225} C_VEL
LIN {X 0,Y 531.004,Z 458.344,A -85,B 0,C 180,E1 -4526.744,E2 -4526.744} C_VEL
LIN {X 0,Y 530.993,Z 458.329,A -85,B 0,C 180,E1 -4529.322,E2 -4529.322} C_VEL
LIN {X 0,Y 530.973,Z 458.331,A -85,B 0,C 180,E1 -4532.104,E2 -4532.104} C_VEL
LIN {X 0,Y 530.986,Z 458.346,A -85,B 0,C 180,E1 -4534.855,E2 -4534.855} C_VEL
LIN {X 0,Y 530.961,Z 458.34,A -85,B 0,C 180,E1 -4537.508,E2 -4537.508} C_VEL
LIN {X 0,Y 530.98,Z 458.331,A -85,B 0,C 180,E1 -4540.433,E2 -4540.433} C_VEL
LIN {X 0,Y 530.962,Z 458.345,A -85,B 0,C 180,E1 -4543.283,E2 -4543.283} C_VEL
LIN {X 0,Y 530.957,Z 458.343,A -85,B 0,C 180,E1 -4543.581,E2 -4543.581} C_VEL
LIN {X 0,Y 530.287,Z 458.426,A -85,B 0,C 180,E1 -4544.214,E2 -4544.214} C_VEL
LIN {X 0,Y 527.441,Z 458.784,A -85,B 0,C 180,E1 -4545.243,E2 -4545.243} C_VEL
LIN {X 0,Y 525.038,Z 459.086,A -85,B 0,C 180,E1 -4546.072,E2 -4546.072} C_VEL
LIN {X 0,Y 524.005,Z 459.211,A -85,B 0,C 180,E1 -4546.711,E2 -4546.711} C_VEL
LIN {X 0,Y 523.92,Z 459.219,A -85,B 0,C 180,E1 -4546.928,E2 -4546.928} C_VEL
LIN {X 0,Y 523.945,Z 459.215,A -85,B 0,C 180,E1 -4549.921,E2 -4549.921} C_VEL
LIN {X 0,Y 523.909,Z 459.222,A -85,B 0,C 180,E1 -4552.869,E2 -4552.869} C_VEL
LIN {X 0,Y 523.94,Z 459.202,A -85,B 0,C 180,E1 -4555.711,E2 -4555.711} C_VEL
LIN {X 0,Y 523.931,Z 459.217,A -85,B 0,C 180,E1 -4558.457,E2 -4558.457} C_VEL
LIN {X 0,Y 523.939,Z 459.219,A -85,B 0,C 180,E1 -4561.126,E2 -4561.126} C_VEL
LIN {X 0,Y 523.985,Z 459.207,A -85,B 0,C 180,E1 -4563.981,E2 -4563.981} C_VEL
LIN {X 0,Y 523.928,Z 459.218,A -85,B 0,C 180,E1 -4566.271,E2 -4566.271} C_VEL
LIN {X 0,Y 523.948,Z 459.214,A -85,B 0,C 180,E1 -4568.767,E2 -4568.767} C_VEL
LIN {X 0,Y 523.954,Z 459.207,A -85,B 0,C 180,E1 -4571.221,E2 -4571.221} C_VEL
LIN {X 0,Y 523.936,Z 459.198,A -85,B 0,C 180,E1 -4573.639,E2 -4573.639} C_VEL
LIN {X 0,Y 524.02,Z 459.411,A -85,B 0,C 180,E1 -4575.156,E2 -4575.156} C_VEL
LIN {X 0,Y 524.297,Z 460.441,A -85,B 0,C 180,E1 -4575.279,E2 -4575.279} C_VEL
LIN {X 0,Y 525.914,Z 465.216,A -85,B 0,C 180,E1 -4575.405,E2 -4575.405} C_VEL
LIN {X 0,Y 525.729,Z 539.361,A -85,B 0,C 180,E1 -4576.446,E2 -4576.446} C_VEL
LIN {X 0,Y 525.657,Z 552.48,A -85,B 0,C 180,E1 -4576.789,E2 -4576.789} C_VEL
LIN {X 0,Y 525.466,Z 564.173,A -85,B 0,C 180,E1 -4577.236,E2 -4577.236} C_VEL
LIN {X 0,Y 525.312,Z 575.912,A -85,B 0,C 180,E1 -4577.842,E2 -4577.842} C_VEL
LIN {X 0,Y 524.994,Z 587.395,A -85,B 0,C 180,E1 -4578.612,E2 -4578.612} C_VEL
LIN {X 0,Y 524.724,Z 597.746,A -85,B 0,C 180,E1 -4579.485,E2 -4579.485} C_VEL
LIN {X 0,Y 524.466,Z 606.192,A -85,B 0,C 180,E1 -4580.358,E2 -4580.358} C_VEL
LIN {X 0,Y 524.3,Z 613.946,A -85,B 0,C 180,E1 -4581.327,E2 -4581.327} C_VEL
LIN {X 0,Y 524.05,Z 621.642,A -85,B 0,C 180,E1 -4582.506,E2 -4582.506} C_VEL
LIN {X 0,Y 523.921,Z 628.459,A -85,B 0,C 180,E1 -4583.84,E2 -4583.84} C_VEL
LIN {X 0,Y 523.696,Z 633.092,A -85,B 0,C 180,E1 -4584.996,E2 -4584.996} C_VEL
LIN {X 0,Y 523.665,Z 636.618,A -85,B 0,C 180,E1 -4586.152,E2 -4586.152} C_VEL
LIN {X 0,Y 523.61,Z 638.445,A -85,B 0,C 180,E1 -4586.922,E2 -4586.922} C_VEL
LIN {X 0,Y 523.586,Z 639.822,A -85,B 0,C 180,E1 -4587.692,E2 -4587.692} C_VEL
LIN {X 0,Y 523.555,Z 641.402,A -85,B 0,C 180,E1 -4589.231,E2 -4589.231} C_VEL
LIN {X 0,Y 523.546,Z 641.636,A -85,B 0,C 180,E1 -4590,E2 -4590} C_VEL
LIN {X 0,Y 523.555,Z 641.456,A -85,B 0,C 180,E1 -4590.769,E2 -4590.769} C_VEL
LIN {X 0,Y 523.585,Z 639.946,A -85,B 0,C 180,E1 -4592.308,E2 -4592.308} C_VEL
LIN {X 0,Y 523.608,Z 638.625,A -85,B 0,C 180,E1 -4593.078,E2 -4593.078} C_VEL
LIN {X 0,Y 523.719,Z 635.82,A -85,B 0,C 180,E1 -4594.233,E2 -4594.233} C_VEL
LIN {X 0,Y 523.794,Z 632.023,A -85,B 0,C 180,E1 -4595.389,E2 -4595.389} C_VEL
LIN {X 0,Y 523.881,Z 626.897,A -85,B 0,C 180,E1 -4596.596,E2 -4596.596} C_VEL
LIN {X 0,Y 524.108,Z 619.729,A -85,B 0,C 180,E1 -4597.9,E2 -4597.9} C_VEL
LIN {X 0,Y 524.375,Z 611.714,A -85,B 0,C 180,E1 -4599.06,E2 -4599.06} C_VEL
LIN {X 0,Y 524.561,Z 603.505,A -85,B 0,C 180,E1 -4600.03,E2 -4600.03} C_VEL
LIN {X 0,Y 524.897,Z 593.331,A -85,B 0,C 180,E1 -4600.999,E2 -4600.999} C_VEL
LIN {X 0,Y 525.191,Z 582.997,A -85,B 0,C 180,E1 -4601.792,E2 -4601.792} C_VEL
LIN {X 0,Y 525.35,Z 571.114,A -85,B 0,C 180,E1 -4602.518,E2 -4602.518} C_VEL
LIN {X 0,Y 525.534,Z 558.602,A -85,B 0,C 180,E1 -4603.086,E2 -4603.086} C_VEL
LIN {X 0,Y 525.702,Z 545.469,A -85,B 0,C 180,E1 -4603.505,E2 -4603.505} C_VEL
LIN {X 0,Y 525.781,Z 533.027,A -85,B 0,C 180,E1 -4603.749,E2 -4603.749} C_VEL
LIN {X 0,Y 525.969,Z 465.316,A -85,B 0,C 180,E1 -4604.682,E2 -4604.682} C_VEL
LIN {X 0,Y 524.135,Z 459.984,A -85,B 0,C 180,E1 -4604.844,E2 -4604.844} C_VEL
LIN {X 0,Y 524.023,Z 459.285,A -85,B 0,C 180,E1 -4604.98,E2 -4604.98} C_VEL
LIN {X 0,Y 523.966,Z 459.196,A -85,B 0,C 180,E1 -4607.968,E2 -4607.968} C_VEL
LIN {X 0,Y 523.974,Z 459.215,A -85,B 0,C 180,E1 -4610.409,E2 -4610.409} C_VEL
LIN {X 0,Y 523.912,Z 459.219,A -85,B 0,C 180,E1 -4612.893,E2 -4612.893} C_VEL
LIN {X 0,Y 523.953,Z 459.214,A -85,B 0,C 180,E1 -4615.418,E2 -4615.418} C_VEL
LIN {X 0,Y 523.968,Z 459.205,A -85,B 0,C 180,E1 -4617.998,E2 -4617.998} C_VEL
LIN {X 0,Y 523.947,Z 459.223,A -85,B 0,C 180,E1 -4620.855,E2 -4620.855} C_VEL
LIN {X 0,Y 523.959,Z 459.214,A -85,B 0,C 180,E1 -4623.734,E2 -4623.734} C_VEL
LIN {X 0,Y 523.918,Z 459.218,A -85,B 0,C 180,E1 -4626.403,E2 -4626.403} C_VEL
LIN {X 0,Y 523.922,Z 459.227,A -85,B 0,C 180,E1 -4629.083,E2 -4629.083} C_VEL
LIN {X 0,Y 523.954,Z 459.209,A -85,B 0,C 180,E1 -4632.117,E2 -4632.117} C_VEL
LIN {X 0,Y 523.952,Z 459.221,A -85,B 0,C 180,E1 -4635.308,E2 -4635.308} C_VEL
LIN {X 0,Y 523.957,Z 459.214,A -85,B 0,C 180,E1 -4638.688,E2 -4638.688} C_VEL
LIN {X 0,Y 523.912,Z 459.217,A -85,B 0,C 180,E1 -4641.898,E2 -4641.898} C_VEL
LIN {X 0,Y 523.934,Z 459.222,A -85,B 0,C 180,E1 -4644.908,E2 -4644.908} C_VEL
LIN {X 0,Y 523.936,Z 459.209,A -85,B 0,C 180,E1 -4647.677,E2 -4647.677} C_VEL
LIN {X 0,Y 523.963,Z 459.204,A -85,B 0,C 180,E1 -4650.673,E2 -4650.673} C_VEL
LIN {X 0,Y 523.97,Z 459.214,A -85,B 0,C 180,E1 -4653.728,E2 -4653.728} C_VEL
LIN {X 0,Y 523.928,Z 459.216,A -85,B 0,C 180,E1 -4656.27,E2 -4656.27} C_VEL
LIN {X 0,Y 523.939,Z 459.215,A -85,B 0,C 180,E1 -4658.766,E2 -4658.766} C_VEL
LIN {X 0,Y 523.945,Z 459.223,A -85,B 0,C 180,E1 -4661.22,E2 -4661.22} C_VEL
LIN {X 0,Y 523.931,Z 459.217,A -85,B 0,C 180,E1 -4663.639,E2 -4663.639} C_VEL
LIN {X 0,Y 523.936,Z 459.217,A -85,B 0,C 180,E1 -4666.028,E2 -4666.028} C_VEL
LIN {X 0,Y 524.002,Z 459.207,A -85,B 0,C 180,E1 -4668.394,E2 -4668.394} C_VEL
LIN {X 0,Y 523.999,Z 459.214,A -85,B 0,C 180,E1 -4671.516,E2 -4671.516} C_VEL
LIN {X 0,Y 524.077,Z 459.198,A -85,B 0,C 180,E1 -4674.614,E2 -4674.614} C_VEL
LIN {X 0,Y 524.103,Z 459.197,A -85,B 0,C 180,E1 -4677.694,E2 -4677.694} C_VEL
LIN {X 0,Y 524.116,Z 459.193,A -85,B 0,C 180,E1 -4680.768,E2 -4680.768} C_VEL
LIN {X 0,Y 524.067,Z 459.201,A -85,B 0,C 180,E1 -4683.075,E2 -4683.075} C_VEL
LIN {X 0,Y 524.037,Z 459.204,A -85,B 0,C 180,E1 -4686.159,E2 -4686.159} C_VEL
LIN {X 0,Y 523.994,Z 459.214,A -85,B 0,C 180,E1 -4689.262,E2 -4689.262} C_VEL
LIN {X 0,Y 523.998,Z 459.213,A -85,B 0,C 180,E1 -4691.743,E2 -4691.743} C_VEL
LIN {X 0,Y 523.982,Z 459.213,A -85,B 0,C 180,E1 -4695.053,E2 -4695.053} C_VEL
LIN {X 0,Y 523.955,Z 459.208,A -85,B 0,C 180,E1 -4697.969,E2 -4697.969} C_VEL
LIN {X 0,Y 523.963,Z 459.209,A -85,B 0,C 180,E1 -4700.41,E2 -4700.41} C_VEL
LIN {X 0,Y 523.908,Z 459.22,A -85,B 0,C 180,E1 -4702.894,E2 -4702.894} C_VEL
LIN {X 0,Y 523.947,Z 459.22,A -85,B 0,C 180,E1 -4705.419,E2 -4705.419} C_VEL
LIN {X 0,Y 523.963,Z 459.216,A -85,B 0,C 180,E1 -4707.999,E2 -4707.999} C_VEL
LIN {X 0,Y 523.945,Z 459.215,A -85,B 0,C 180,E1 -4710.857,E2 -4710.857} C_VEL
LIN {X 0,Y 523.956,Z 459.218,A -85,B 0,C 180,E1 -4713.736,E2 -4713.736} C_VEL
LIN {X 0,Y 523.916,Z 459.219,A -85,B 0,C 180,E1 -4716.405,E2 -4716.405} C_VEL
LIN {X 0,Y 523.918,Z 459.218,A -85,B 0,C 180,E1 -4719.085,E2 -4719.085} C_VEL
LIN {X 0,Y 523.951,Z 459.214,A -85,B 0,C 180,E1 -4722.119,E2 -4722.119} C_VEL
LIN {X 0,Y 523.951,Z 459.211,A -85,B 0,C 180,E1 -4725.309,E2 -4725.309} C_VEL
LIN {X 0,Y 523.969,Z 459.209,A -85,B 0,C 180,E1 -4728.688,E2 -4728.688} C_VEL
LIN {X 0,Y 523.923,Z 459.218,A -85,B 0,C 180,E1 -4731.08,E2 -4731.08} C_VEL
LIN {X 0,Y 523.921,Z 459.221,A -85,B 0,C 180,E1 -4733.828,E2 -4733.828} C_VEL
LIN {X 0,Y 523.94,Z 459.216,A -85,B 0,C 180,E1 -4736.636,E2 -4736.636} C_VEL
LIN {X 0,Y 523.956,Z 459.208,A -85,B 0,C 180,E1 -4739.357,E2 -4739.357} C_VEL
LIN {X 0,Y 524.015,Z 459.427,A -85,B 0,C 180,E1 -4741.459,E2 -4741.459} C_VEL
LIN {X 0,Y 526.485,Z 471.054,A -85,B 0,C 180,E1 -4743.009,E2 -4743.009} C_VEL
LIN {X 0,Y 526.289,Z 486.7,A -85,B 0,C 180,E1 -4744.886,E2 -4744.886} C_VEL
LIN {X 0,Y 525.802,Z 508.759,A -85,B 0,C 180,E1 -4747.487,E2 -4747.487} C_VEL
LIN {X 0,Y 525.324,Z 532.528,A -85,B 0,C 180,E1 -4750.257,E2 -4750.257} C_VEL
LIN {X 0,Y 524.839,Z 558.723,A -85,B 0,C 180,E1 -4753.268,E2 -4753.268} C_VEL
LIN {X 0,Y 524.636,Z 572.46,A -85,B 0,C 180,E1 -4754.817,E2 -4754.817} C_VEL
LIN {X 0,Y 525.973,Z 584.449,A -85,B 0,C 180,E1 -4755.033,E2 -4755.033} C_VEL
LIN {X 0,Y 525.513,Z 682.827,A -85,B 0,C 180,E1 -4756.392,E2 -4756.392} C_VEL
LIN {X 0,Y 525.271,Z 696.182,A -85,B 0,C 180,E1 -4756.73,E2 -4756.73} C_VEL
LIN {X 0,Y 525.05,Z 709.594,A -85,B 0,C 180,E1 -4757.241,E2 -4757.241} C_VEL
LIN {X 0,Y 524.78,Z 721.487,A -85,B 0,C 180,E1 -4757.861,E2 -4757.861} C_VEL
LIN {X 0,Y 524.518,Z 733.949,A -85,B 0,C 180,E1 -4758.699,E2 -4758.699} C_VEL
LIN {X 0,Y 524.208,Z 744.304,A -85,B 0,C 180,E1 -4759.573,E2 -4759.573} C_VEL
LIN {X 0,Y 523.975,Z 753.642,A -85,B 0,C 180,E1 -4760.543,E2 -4760.543} C_VEL
LIN {X 0,Y 523.759,Z 762.669,A -85,B 0,C 180,E1 -4761.706,E2 -4761.706} C_VEL
LIN {X 0,Y 523.583,Z 769.849,A -85,B 0,C 180,E1 -4762.868,E2 -4762.868} C_VEL
LIN {X 0,Y 523.544,Z 776.367,A -85,B 0,C 180,E1 -4764.222,E2 -4764.222} C_VEL
LIN {X 0,Y 523.361,Z 780.677,A -85,B 0,C 180,E1 -4765.379,E2 -4765.379} C_VEL
LIN {X 0,Y 523.443,Z 782.958,A -85,B 0,C 180,E1 -4766.151,E2 -4766.151} C_VEL
LIN {X 0,Y 523.367,Z 784.807,A -85,B 0,C 180,E1 -4766.921,E2 -4766.921} C_VEL
LIN {X 0,Y 523.334,Z 786.193,A -85,B 0,C 180,E1 -4767.691,E2 -4767.691} C_VEL
LIN {X 0,Y 523.25,Z 787.785,A -85,B 0,C 180,E1 -4769.23,E2 -4769.23} C_VEL
LIN {X 0,Y 523.246,Z 788,A -85,B 0,C 180,E1 -4770,E2 -4770} C_VEL
LIN {X 0,Y 523.274,Z 787.183,A -85,B 0,C 180,E1 -4771.539,E2 -4771.539} C_VEL
LIN {X 0,Y 523.334,Z 786.196,A -85,B 0,C 180,E1 -4772.309,E2 -4772.309} C_VEL
LIN {X 0,Y 523.367,Z 784.81,A -85,B 0,C 180,E1 -4773.079,E2 -4773.079} C_VEL
LIN {X 0,Y 523.441,Z 781.895,A -85,B 0,C 180,E1 -4774.235,E2 -4774.235} C_VEL
LIN {X 0,Y 523.464,Z 777.948,A -85,B 0,C 180,E1 -4775.393,E2 -4775.393} C_VEL
LIN {X 0,Y 523.523,Z 772.727,A -85,B 0,C 180,E1 -4776.581,E2 -4776.581} C_VEL
LIN {X 0,Y 523.665,Z 766.466,A -85,B 0,C 180,E1 -4777.713,E2 -4777.713} C_VEL
LIN {X 0,Y 523.852,Z 758.413,A -85,B 0,C 180,E1 -4778.875,E2 -4778.875} C_VEL
LIN {X 0,Y 524.079,Z 750.114,A -85,B 0,C 180,E1 -4779.845,E2 -4779.845} C_VEL
LIN {X 0,Y 524.321,Z 739.971,A -85,B 0,C 180,E1 -4780.816,E2 -4780.816} C_VEL
LIN {X 0,Y 524.644,Z 728.455,A -85,B 0,C 180,E1 -4781.696,E2 -4781.696} C_VEL
LIN {X 0,Y 524.881,Z 717.376,A -85,B 0,C 180,E1 -4782.37,E2 -4782.37} C_VEL
LIN {X 0,Y 525.111,Z 705.025,A -85,B 0,C 180,E1 -4782.954,E2 -4782.954} C_VEL
LIN {X 0,Y 525.338,Z 692.103,A -85,B 0,C 180,E1 -4783.391,E2 -4783.391} C_VEL
LIN {X 0,Y 525.527,Z 678.453,A -85,B 0,C 180,E1 -4783.682,E2 -4783.682} C_VEL
LIN {X 0,Y 525.813,Z 581.818,A -85,B 0,C 180,E1 -4785.008,E2 -4785.008} C_VEL
LIN {X 0,Y 524.619,Z 572.322,A -85,B 0,C 180,E1 -4785.191,E2 -4785.191} C_VEL
